# B&R Automation Studio project VInRoS_BaR_AS_Program (part 2)

#### Main.c
```c
#include <bur/plctypes.h>
#include <standard.h>

#ifdef _DEFAULT_INCLUDES
#include <AsDefault.h>
#endif

#include "Main.h"

_LOCAL struct MpAxisBasic MpAxisBasic_0;
_LOCAL struct MpAxisBasicParType AxisParameters;
_LOCAL enum Mechanism_State_ID_enum state_id;

void _INIT ProgramInit(void)
{
	memset(&Global_VInRoS_Str.Mech_Id_3, 0, sizeof(Global_VInRoS_Str.Mech_Id_3));

	MpAxisBasic_0.Enable     = 1;
	MpAxisBasic_0.MpLink     = &gAxis_Mech_03;
	MpAxisBasic_0.Parameters = &AxisParameters;

	Trajectory_Str.Targets.Position[0] = 700.0;
	Trajectory_Str.Targets.Position[1] = 100.0;
	Trajectory_Str.Targets.Position[2] = 400.0;
	Trajectory_Str.Targets.Position[3] = 600.0;
	Trajectory_Str.Targets.Position[4] = 300.0;

	Trajectory_Str.Targets.Velocity[0] = 400.0;
	Trajectory_Str.Targets.Velocity[1] = 200.0;
	Trajectory_Str.Targets.Velocity[2] = 400.0;
	Trajectory_Str.Targets.Velocity[3] = 100.0;
	Trajectory_Str.Targets.Velocity[4] = 400.0;

	Trajectory_Str.Length = 5;

	state_id = MECH_STATE_ACTIVE;
}

void _CYCLIC ProgramCyclic(void)
{
	switch(state_id){
		case MECH_STATE_ACTIVE:
			{
				if(Global_VInRoS_Str.Mech_Id_3.Info.Active == 1){
					state_id = MECH_STATE_POWER;
				}
			}
			break;

		case MECH_STATE_POWER:
			{
				if(Global_VInRoS_Str.Mech_Id_3.Info.Power == 1){
					state_id = MECH_STATE_HOME;
				}
			}
			break;

		case MECH_STATE_HOME:
			{
				if(Global_VInRoS_Str.Mech_Id_3.Info.Home == 1){
					MpAxisBasic_0.Home = 0;
					Global_VInRoS_Str.Mech_Id_3.Command.Home = 0;
					state_id = MECH_STATE_WAIT;
				}
			}
			break;

		case MECH_STATE_WAIT:
			{
				if(Global_VInRoS_Str.Mech_Id_3.Command.Home == 1){
					state_id = MECH_STATE_HOME_UPD_PARAMETERS;
				}

				if(Global_VInRoS_Str.Mech_Id_3.Command.Start == 1){
					Trajectory_Str.Iteration = 0;
					state_id = MECH_STATE_UPD_PARAMETERS;
				}
			}
			break;

		case MECH_STATE_UPD_PARAMETERS:
			{
				Global_VInRoS_Str.Mech_Id_3.Parameters.Position = Trajectory_Str.Targets.Position[Trajectory_Str.Iteration];
				Global_VInRoS_Str.Mech_Id_3.Parameters.Velocity = Trajectory_Str.Targets.Velocity[Trajectory_Str.Iteration];
				Global_VInRoS_Str.Mech_Id_3.Parameters.Acc_Dec  = Trajectory_Str.Targets.Velocity[Trajectory_Str.Iteration]*10;

				Global_VInRoS_Str.Mech_Id_3.Command.Update = 1;
				if(Global_VInRoS_Str.Mech_Id_3.Info.Update_Done == 1){
					state_id = MECH_STATE_MOTION_1;
				}
			}
			break;

		case MECH_STATE_MOTION_1:
			{
				Global_VInRoS_Str.Mech_Id_3.Command.Move = 1;
				if(Global_VInRoS_Str.Mech_Id_3.Info.Move_Active == 1){
					state_id = MECH_STATE_MOTION_2;
				}
			}
			break;

		case MECH_STATE_MOTION_2:
			{
				if(Global_VInRoS_Str.Mech_Id_3.Command.Stop == 1){
					state_id = MECH_STATE_STOP;
				}else{
					if(Global_VInRoS_Str.Mech_Id_3.Info.In_Position == 1){
						Global_VInRoS_Str.Mech_Id_3.Command.Move = 0;

						if(Trajectory_Str.Iteration == Trajectory_Str.Length - 1){
							state_id = MECH_STATE_WAIT;
						}else{
							Trajectory_Str.Iteration++;
							state_id = MECH_STATE_UPD_PARAMETERS;
						}
					}
				}
			}
			break;

		case MECH_STATE_HOME_UPD_PARAMETERS:
			{
				Global_VInRoS_Str.Mech_Id_3.Parameters.Position = 400.0;
				Global_VInRoS_Str.Mech_Id_3.Parameters.Velocity = 250.0;
				Global_VInRoS_Str.Mech_Id_3.Parameters.Acc_Dec  = 2500.0;

				Global_VInRoS_Str.Mech_Id_3.Command.Update = 1;
				if(Global_VInRoS_Str.Mech_Id_3.Info.Update_Done == 1){
					state_id = MECH_STATE_HOME_MOTION_1;
				}
			}
			break;

		case MECH_STATE_HOME_MOTION_1:
			{
				Global_VInRoS_Str.Mech_Id_3.Command.Move = 1;
				if(Global_VInRoS_Str.Mech_Id_3.Info.Move_Active == 1){
					state_id = MECH_STATE_HOME_MOTION_2;
				}
			}
			break;

		case MECH_STATE_HOME_MOTION_2:
			{
				if(Global_VInRoS_Str.Mech_Id_3.Info.In_Position == 1){
					Global_VInRoS_Str.Mech_Id_3.Command.Move = 0;
					Global_VInRoS_Str.Mech_Id_3.Command.Home = 0;
					state_id = MECH_STATE_WAIT;
				}
			}
			break;

		case MECH_STATE_STOP:
			{
				Global_VInRoS_Str.Mech_Id_3.Command.Stop  = 0;
				Global_VInRoS_Str.Mech_Id_3.Command.Start = 0;

				Global_VInRoS_Str.Mech_Id_3.Command.Move = 0;
				if(Global_VInRoS_Str.Mech_Id_3.Info.Move_Active == 0){
					state_id = MECH_STATE_WAIT;
				}
			}
			break;

		case MECH_STATE_SAFETY:
			{
			}
			break;

		case MECH_STATE_ERROR:
			{
				Global_VInRoS_Str.Mech_Id_3.Command.Home   = 0;
				Global_VInRoS_Str.Mech_Id_3.Command.Update = 0;
				Global_VInRoS_Str.Mech_Id_3.Command.Stop   = 0;
				Global_VInRoS_Str.Mech_Id_3.Command.Start  = 0;
				Global_VInRoS_Str.Mech_Id_3.Command.Move   = 0;

				Global_VInRoS_Str.Mech_Id_3.Command.Move = 0;
				if(Global_VInRoS_Str.Mech_Id_3.Info.Error == 0){
					state_id = MECH_STATE_WAIT;
				}
			}
			break;

	}

	AxisParameters.Position     = Global_VInRoS_Str.Mech_Id_3.Parameters.Position;
	AxisParameters.Velocity     = Global_VInRoS_Str.Mech_Id_3.Parameters.Velocity;
	AxisParameters.Acceleration = Global_VInRoS_Str.Mech_Id_3.Parameters.Acc_Dec;
	AxisParameters.Deceleration = Global_VInRoS_Str.Mech_Id_3.Parameters.Acc_Dec;

	MpAxisBasic_0.Power = Global_VInRoS_Str.Mech_Id_3.Command.Power;
	if(Global_VInRoS_Str.Mech_Id_3.Command.Home == 1 && Global_VInRoS_Str.Mech_Id_3.Info.Home == 0){
		MpAxisBasic_0.Home = 1;
	}
	MpAxisBasic_0.ErrorReset = Global_VInRoS_Str.Mech_Id_3.Command.Reset_Error;
	MpAxisBasic_0.Update     = Global_VInRoS_Str.Mech_Id_3.Command.Update;
	MpAxisBasic_0.MoveAbsolute = Global_VInRoS_Str.Mech_Id_3.Command.Move;

	MpAxisBasic(&MpAxisBasic_0);

	Global_VInRoS_Str.Mech_Id_3.Info.Active = MpAxisBasic_0.Active;
	Global_VInRoS_Str.Mech_Id_3.Info.Power  = MpAxisBasic_0.PowerOn;
	Global_VInRoS_Str.Mech_Id_3.Info.Home   = MpAxisBasic_0.IsHomed;
	Global_VInRoS_Str.Mech_Id_3.Info.Error  = MpAxisBasic_0.Error;
	Global_VInRoS_Str.Mech_Id_3.Info.Update_Done = MpAxisBasic_0.UpdateDone;
	Global_VInRoS_Str.Mech_Id_3.Info.Move_Active = MpAxisBasic_0.MoveActive;
	if(MpAxisBasic_0.InPosition == 1 && MpAxisBasic_0.MoveDone == 1){
		Global_VInRoS_Str.Mech_Id_3.Info.In_Position = 1;
	}else{
		Global_VInRoS_Str.Mech_Id_3.Info.In_Position = 0;
	}
	Global_VInRoS_Str.Mech_Id_3.Position = MpAxisBasic_0.Position;

	if(Global_VInRoS_Str.Mech_Id_3.Info.Error == 1){
		state_id = MECH_STATE_ERROR;
	}

	if(SAFETY_ACTIVE == 0 || SAFETY_STATUS == 0){
		Global_VInRoS_Str.Mech_Id_3.Info.Safety = 1;
	}else{
		Global_VInRoS_Str.Mech_Id_3.Info.Safety = 0;
	}
	if(SAFETY_ACTIVE == 1 || SAFETY_STATUS == 0){
		RESET_SAFETY = Global_VInRoS_Str.Mech_Id_3.Command.Reset_Safety;
	}
}
```

### Program Logical/T_EX600 (ANSIC)

#### Main.h
```c
#include <bur/plctypes.h>

#ifdef _DEFAULT_INCLUDES
	#include <AsDefault.h>
#endif

typedef enum EX600_State_ID_enum{
	EX600_STATE_ACTIVE,
	EX600_STATE_HOME,
	EX600_STATE_WAIT,
	EX600_STATE_ERROR
}EX600_State_ID_enum;
```

#### Main.c
```c
// Include B&R Automation libraries (declarations for B&R ANSI C extensions).
#include <bur/plctypes.h>

#ifdef _DEFAULT_INCLUDES
	#include <AsDefault.h>
#endif

#include <Main.h>

// Custom Lib.: Base conversion between data.
#include <Converter.h>

/*  Local Variables.  */
_LOCAL enum EX600_State_ID_enum state_id;

_LOCAL struct Convert_BOOL_Array_To_USINT C_BOOL_Arr_To_USINT_1;
_LOCAL struct Convert_USINT_To_BOOL_Array C_USINT_To_BOOL_Arr_1;
_LOCAL struct Convert_USINT_To_BOOL_Array C_USINT_To_BOOL_Arr_2;

/**
 * Program Intitialization
 */
void _INIT ProgramInit(void)
{
	memset(&Global_VInRoS_Str.EX_600, 0, sizeof(Global_VInRoS_Str.EX_600));

	state_id = EX600_STATE_ACTIVE;
}

/**
 * Program Cyclic
 *
 * Duration (Cycle Time): 10000 [ms]
 * Tolerance            : 10000 [ms]
 */
void _CYCLIC ProgramCyclic(void)
{
	switch(state_id){
		case EX600_STATE_ACTIVE:
			{
				if(Global_VInRoS_Str.EX_600.Slave.Info.Active == 1){
					state_id = EX600_STATE_HOME;
				}
			}
			break;

		case EX600_STATE_HOME:
			{
				if(Global_VInRoS_Str.EX_600.Slave.Command.Home == 1){
					memset(C_BOOL_Arr_To_USINT_1.INPUT, 0, sizeof(C_BOOL_Arr_To_USINT_1.INPUT));
					C_USINT_To_BOOL_Arr_1.INPUT = 0;
					C_USINT_To_BOOL_Arr_2.INPUT = 0;

					Global_VInRoS_Str.EX_600.Slave.Info.Home = 1;
					Global_VInRoS_Str.EX_600.Slave.Command.Home = 0;
					state_id = EX600_STATE_WAIT;
				}
			}
			break;

		case EX600_STATE_WAIT:
			{
				int i;
				for(i = 0; i < (int)(sizeof(C_BOOL_Arr_To_USINT_1.INPUT)/sizeof(C_BOOL_Arr_To_USINT_1.INPUT[0])); i++){
					C_BOOL_Arr_To_USINT_1.INPUT[i] = Global_VInRoS_Str.EX_600.Slave.Output[i];
				}
				Convert_BOOL_Array_To_USINT(&C_BOOL_Arr_To_USINT_1);

				Convert_USINT_To_BOOL_Array(&C_USINT_To_BOOL_Arr_1);
				int j;
				for(j = 0; j < (int)(sizeof(C_USINT_To_BOOL_Arr_1.OUTPUT)/sizeof(C_USINT_To_BOOL_Arr_1.OUTPUT[0])); j++){
					Global_VInRoS_Str.EX_600.Slave.Input[j] = C_USINT_To_BOOL_Arr_1.OUTPUT[j];
				}
				Convert_USINT_To_BOOL_Array(&C_USINT_To_BOOL_Arr_2);
				int k;
				for(k = 0; k < (int)(sizeof(C_USINT_To_BOOL_Arr_2.OUTPUT)/sizeof(C_USINT_To_BOOL_Arr_2.OUTPUT[0])); k++){
					Global_VInRoS_Str.EX_600.Slave.Input[k + 8] = C_USINT_To_BOOL_Arr_2.OUTPUT[k];
				}

			}
			break;

		case EX600_STATE_ERROR:
			{
				if(Global_VInRoS_Str.EX_600.Slave.Info.Error == 0){
					state_id = EX600_STATE_WAIT;
				}
			}
			break;
	}

	if(Global_VInRoS_Str.EX_600.Slave.Info.Error == 1){
		state_id = EX600_STATE_ERROR;
	}
}
```

### Program Logical/T_ROB_1 (ANSIC)

#### Main.c - Init, cyclic, exit code
```c
#include <bur/plctypes.h>

#ifdef _DEFAULT_INCLUDES
#include <AsDefault.h>
#endif

#include <Main.h>

_LOCAL enum Robot_State_ID_enum state_id;

/*
if(Global_VInRoS_Str.Rob_Id_1.Command.Start == TRUE){
	ABB_Library_Rob_1.Command.ID.Motion = MAIN_ID_JOINT_ABSOLUTE;
	ABB_Library_Rob_1.Command.START = TRUE;
	Global_VInRoS_Str.Rob_Id_1.Command.Start = FALSE;
}
   */

/*
if(Global_VInRoS_Str.Rob_Id_1.Command.STOP == TRUE){
	ABB_Library_Rob_1.Command.STOP = TRUE;
	Global_VInRoS_Str.Rob_Id_1.Command.STOP = FALSE;
}
*/

void _INIT ProgramInit(void)
{
	memset(&Global_VInRoS_Str.Rob_Id_1, 0, sizeof(Global_VInRoS_Str.Rob_Id_1));

	ABB_Library_Rob_1.Enable = TRUE;

	//
	ABB_Library_Rob_1.Rob_Tool.robHold = FALSE;
	ABB_Library_Rob_1.Rob_Tool.tFrame.Position[0] = 0.0; ABB_Library_Rob_1.Rob_Tool.tFrame.Position[1] = 0.0;
	ABB_Library_Rob_1.Rob_Tool.tFrame.Position[2] = 0.0;
	ABB_Library_Rob_1.Rob_Tool.tFrame.Rotation[0] = 1.0; ABB_Library_Rob_1.Rob_Tool.tFrame.Rotation[1] = 0.0;
	ABB_Library_Rob_1.Rob_Tool.tFrame.Rotation[2] = 0.0; ABB_Library_Rob_1.Rob_Tool.tFrame.Rotation[3] = 0.0;
	ABB_Library_Rob_1.Rob_Tool.tLoad.mass = 0.0;
	ABB_Library_Rob_1.Rob_Tool.tLoad.center_of_gravity[0] = 0.0; ABB_Library_Rob_1.Rob_Tool.tLoad.center_of_gravity[1] = 0.0;
	ABB_Library_Rob_1.Rob_Tool.tLoad.center_of_gravity[2] = 0.0;
	ABB_Library_Rob_1.Rob_Tool.tLoad.intertial_axes[0] = 1.0; ABB_Library_Rob_1.Rob_Tool.tLoad.intertial_axes[1] = 0.0;
	ABB_Library_Rob_1.Rob_Tool.tLoad.intertial_axes[2] = 0.0; ABB_Library_Rob_1.Rob_Tool.tLoad.intertial_axes[3] = 0.0;
	ABB_Library_Rob_1.Rob_Tool.tLoad.moment_of_inertia[0] = 0.0; ABB_Library_Rob_1.Rob_Tool.tLoad.moment_of_inertia[1] = 0.0;
	ABB_Library_Rob_1.Rob_Tool.tLoad.moment_of_inertia[2] = 0.0;

	ABB_Library_Rob_1.Parameter.Joint[0].Q[0] = 130.0; ABB_Library_Rob_1.Parameter.Joint[0].Q[1] = -10.0;
	ABB_Library_Rob_1.Parameter.Joint[0].Q[2] = 15.0; ABB_Library_Rob_1.Parameter.Joint[0].Q[3] = -50.0;
	ABB_Library_Rob_1.Parameter.Joint[0].Q[4] = 60.0; ABB_Library_Rob_1.Parameter.Joint[0].Q[5] = 60.0;
	ABB_Library_Rob_1.Parameter.Speed[0] = vSPEED_100;
	ABB_Library_Rob_1.Parameter.Zone[0]  = zZone_fine;

	ABB_Library_Rob_1.Parameter.Joint[1].Q[0] = 110.0; ABB_Library_Rob_1.Parameter.Joint[1].Q[1] = 60.0;
	ABB_Library_Rob_1.Parameter.Joint[1].Q[2] = -20.0; ABB_Library_Rob_1.Parameter.Joint[1].Q[3] = 0.0;
	ABB_Library_Rob_1.Parameter.Joint[1].Q[4] = -60.0; ABB_Library_Rob_1.Parameter.Joint[1].Q[5] = -40.0;
	ABB_Library_Rob_1.Parameter.Speed[1] = vSPEED_100;
	ABB_Library_Rob_1.Parameter.Zone[1]  = zZone_fine;

	ABB_Library_Rob_1.Parameter.Joint[2].Q[0] = -30.0; ABB_Library_Rob_1.Parameter.Joint[2].Q[1] = 20.0;
	ABB_Library_Rob_1.Parameter.Joint[2].Q[2] = 10.0; ABB_Library_Rob_1.Parameter.Joint[2].Q[3] = 40.0;
	ABB_Library_Rob_1.Parameter.Joint[2].Q[4] = 90.0; ABB_Library_Rob_1.Parameter.Joint[2].Q[5] = 0.0;
	ABB_Library_Rob_1.Parameter.Speed[2] = vSPEED_100;
	ABB_Library_Rob_1.Parameter.Zone[2]  = zZone_fine;

	ABB_Library_Rob_1.Parameter.Joint[3].Q[0] = 0.0; ABB_Library_Rob_1.Parameter.Joint[3].Q[1] = -50.0;
	ABB_Library_Rob_1.Parameter.Joint[3].Q[2] = -20.0; ABB_Library_Rob_1.Parameter.Joint[3].Q[3] = 90.0;
	ABB_Library_Rob_1.Parameter.Joint[3].Q[4] = -40.0; ABB_Library_Rob_1.Parameter.Joint[3].Q[5] = 100.0;
	ABB_Library_Rob_1.Parameter.Speed[3] = vSPEED_100;
	ABB_Library_Rob_1.Parameter.Zone[3]  = zZone_fine;

	ABB_Library_Rob_1.Parameter.Joint[4].Q[0] = 65.0; ABB_Library_Rob_1.Parameter.Joint[4].Q[1] = 10.0;
	ABB_Library_Rob_1.Parameter.Joint[4].Q[2] = 20.0; ABB_Library_Rob_1.Parameter.Joint[4].Q[3] = 50.0;
	ABB_Library_Rob_1.Parameter.Joint[4].Q[4] = 55.0; ABB_Library_Rob_1.Parameter.Joint[4].Q[5] = -20.0;
	ABB_Library_Rob_1.Parameter.Speed[4] = vSPEED_100;
	ABB_Library_Rob_1.Parameter.Zone[4]  = zZone_fine;

	ABB_Library_Rob_1.Parameter.Trajectory_Size = 5;

	/*
	ABB_Library_Rob_1.Parameter.TCP[0].Position[0] = 0.0; ABB_Library_Rob_1.Parameter.TCP[0].Position[1] = 0.0;
	ABB_Library_Rob_1.Parameter.TCP[0].Position[2] = 0.0;
	ABB_Library_Rob_1.Parameter.TCP[0].Rotation[0] = 0.0; ABB_Library_Rob_1.Parameter.TCP[0].Rotation[1] = 0.0;
	ABB_Library_Rob_1.Parameter.TCP[0].Rotation[2] = 0.0;
	ABB_Library_Rob_1.Parameter.TCP[0].Configuration[0] = 0.0; ABB_Library_Rob_1.Parameter.TCP[0].Configuration[1] = 0.0;
	ABB_Library_Rob_1.Parameter.TCP[0].Configuration[2] = 0.0; ABB_Library_Rob_1.Parameter.TCP[0].Configuration[3] = 0.0;
	ABB_Library_Rob_1.Parameter.Speed[0] = 8;
	ABB_Library_Rob_1.Parameter.Zone[0]  = 0;

	ABB_Library_Rob_1.Parameter.Trajectory_Size = 2;
	*/

	/*
	//
	Trajectory_Str.Targets.Position[0].Q[0] = 0.0; Trajectory_Str.Targets.Position[0].Q[1] = 0.0;
	Trajectory_Str.Targets.Position[0].Q[2] = 0.0; Trajectory_Str.Targets.Position[0].Q[3] = 0.0;
	Trajectory_Str.Targets.Position[0].Q[4] = 0.0; Trajectory_Str.Targets.Position[0].Q[5] = 0.0;
	Trajectory_Str.Targets.Speed[0] = 8;
	Trajectory_Str.Targets.Zone[0]  = 0;
	//
	Trajectory_Str.Targets.Position[1].Q[0] = 0.0; Trajectory_Str.Targets.Position[1].Q[1] = 0.0;
	Trajectory_Str.Targets.Position[1].Q[2] = 0.0; Trajectory_Str.Targets.Position[1].Q[3] = 0.0;
	Trajectory_Str.Targets.Position[1].Q[4] = 90.0; Trajectory_Str.Targets.Position[1].Q[5] = 0.0;
	Trajectory_Str.Targets.Speed[1] = 8;
	Trajectory_Str.Targets.Zone[1]  = 0;
	//
	Trajectory_Str.Targets.Position[2].Q[0] = 90.0; Trajectory_Str.Targets.Position[2].Q[1] = 0.0;
	Trajectory_Str.Targets.Position[2].Q[2] = 0.0; Trajectory_Str.Targets.Position[2].Q[3] = 0.0;
	Trajectory_Str.Targets.Position[2].Q[4] = 90.0; Trajectory_Str.Targets.Position[2].Q[5] = 0.0;
	Trajectory_Str.Targets.Speed[2] = 8;
	Trajectory_Str.Targets.Zone[2]  = 0;
	//
	Trajectory_Str.Targets.Position[3].Q[0] = 90.0; Trajectory_Str.Targets.Position[3].Q[1] = 0.0;
	Trajectory_Str.Targets.Position[3].Q[2] = 0.0; Trajectory_Str.Targets.Position[3].Q[3] = 45.0;
	Trajectory_Str.Targets.Position[3].Q[4] = 90.0; Trajectory_Str.Targets.Position[3].Q[5] = 0.0;
	Trajectory_Str.Targets.Speed[3] = 8;
	Trajectory_Str.Targets.Zone[3]  = 0;
	//
	Trajectory_Str.Targets.Position[4].Q[0] = 0.0; Trajectory_Str.Targets.Position[4].Q[1] = 0.0;
	Trajectory_Str.Targets.Position[4].Q[2] = 0.0; Trajectory_Str.Targets.Position[4].Q[3] = 45.0;
	Trajectory_Str.Targets.Position[4].Q[4] = 90.0; Trajectory_Str.Targets.Position[4].Q[5] = 0.0;
	Trajectory_Str.Targets.Speed[4] = 8;
	Trajectory_Str.Targets.Zone[4]  = 0;

	//
	Trajectory_Str.Length = 5;
	*/
}

void _CYCLIC ProgramCyclic(void)
{
	/*
	switch(state_id){
		case ROB_STATE_ACTIVE:
			{
				if(Global_VInRoS_Str.Rob_Id_1.Info.Active == TRUE){
					state_id = ROB_STATE_POWER;
				}
			}
			break;

		case ROB_STATE_POWER:
			{
				if(Global_VInRoS_Str.Rob_Id_1.Info.Power == TRUE){
					state_id = ROB_STATE_WAIT;
				}
			}
			break;

		case ROB_STATE_WAIT:
			{
				Global_VInRoS_Str.Rob_Id_1.Info.Move_Active = FALSE;

				if(Global_VInRoS_Str.Rob_Id_1.Command.Home == TRUE){
					state_id = ROB_STATE_UPD_PARAMETERS;
				}

				if(Global_VInRoS_Str.Rob_Id_1.Command.Start == TRUE){
					Trajectory_Str.Iteration = FALSE;
					state_id = ROB_STATE_HOME_UPD_PARAMETERS;
				}
			}
			break;

		case ROB_STATE_UPD_PARAMETERS:
			{
				memcpy(ABB_Library_Rob_1.Parameter.Position, Trajectory_Str.Targets.Position,
					  (sizeof(Trajectory_Str.Targets.Position) / sizeof(Trajectory_Str.Targets.Position[0])) * sizeof(REAL));
				memcpy(ABB_Library_Rob_1.Parameter.Speed, Trajectory_Str.Targets.Speed,
					   (sizeof(Trajectory_Str.Targets.Speed) / sizeof(Trajectory_Str.Targets.Speed[0])) * sizeof(REAL));
				memcpy(ABB_Library_Rob_1.Parameter.Zone, Trajectory_Str.Targets.Zone,
					   (sizeof(Trajectory_Str.Targets.Zone) / sizeof(Trajectory_Str.Targets.Zone[0])) * sizeof(REAL));

				ABB_Library_Rob_1.Parameter.Trajectory_Size = Trajectory_Str.Length;

				Global_VInRoS_Str.Rob_Id_1.Command.Update = TRUE;

				if(Global_VInRoS_Str.Rob_Id_1.Info.Update_Done == TRUE){
					state_id = ROB_STATE_MOTION_1;
				}
			}
			break;

		case ROB_STATE_MOTION_1:
			{
				Global_VInRoS_Str.Rob_Id_1.Info.Move_Active = TRUE;
			}
			break;

		case ROB_STATE_MOTION_2:
			{

			}
			break;

		case ROB_STATE_HOME_UPD_PARAMETERS:
			{
				Global_VInRoS_Str.Rob_Id_1.Info.Home = FALSE;

				ABB_Library_Rob_1.Parameter.Position[0].Q[0] = 0.0; ABB_Library_Rob_1.Parameter.Position[0].Q[1] = 0.0;
				ABB_Library_Rob_1.Parameter.Position[0].Q[2] = 0.0; ABB_Library_Rob_1.Parameter.Position[0].Q[3] = 0.0;
				ABB_Library_Rob_1.Parameter.Position[0].Q[4] = 0.0; ABB_Library_Rob_1.Parameter.Position[0].Q[5] = 0.0;
				ABB_Library_Rob_1.Parameter.Speed[0] = 5;
				ABB_Library_Rob_1.Parameter.Zone[0]  = 0;

				ABB_Library_Rob_1.Parameter.Trajectory_Size = 1;

				Global_VInRoS_Str.Rob_Id_1.Command.Update = TRUE;

				if(Global_VInRoS_Str.Rob_Id_1.Info.Update_Done == TRUE){
					state_id = ROB_STATE_HOME_MOTION_1;
				}
			}
			break;

		case ROB_STATE_HOME_MOTION_1:
			{

			}
			break;

		case ROB_STATE_HOME_MOTION_2:
			{
				Global_VInRoS_Str.Rob_Id_1.Info.Home = TRUE;
			}
			break;

		case ROB_STATE_STOP:
			{
				Global_VInRoS_Str.Rob_Id_1.Info.Move_Active = FALSE;
			}
			break;

		case ROB_STATE_SAFETY:
			{

			}
			break;

		case ROB_STATE_ERROR:
			{

			}
			break;
	}

	if(Global_VInRoS_Str.Rob_Id_1.Command.Update == TRUE){
		ABB_Library_Rob_1.Command.ID.Update = UPT_ID_TRAJECTORY_JOINT;
		ABB_Library_Rob_1.Command.UPDATE = TRUE;
		Global_VInRoS_Str.Rob_Id_1.Command.Update = FALSE;
	}

	ABB_Library(&ABB_Library_Rob_1);

	Global_VInRoS_Str.Rob_Id_1.Info.Active = ABB_Library_Rob_1.Status.Robot.Active;
	Global_VInRoS_Str.Rob_Id_1.Info.Power = ABB_Library_Rob_1.Status.Robot.System.MOTOR_ON;
	Global_VInRoS_Str.Rob_Id_1.Info.Update_Done = ABB_Library_Rob_1.Status.Robot.Update_Done;
	Global_VInRoS_Str.Rob_Id_1.Info.In_Position = ABB_Library_Rob_1.Status.Robot.In_Position;
	Global_VInRoS_Str.Rob_Id_1.Info.Error  = FALSE;
	Global_VInRoS_Str.Rob_Id_1.Info.Safety = FALSE;

	memcpy(Global_VInRoS_Str.Rob_Id_1.Position.Q, ABB_Library_Rob_1.RT_Data.Q,
		(sizeof(ABB_Library_Rob_1.RT_Data.Q) / sizeof(ABB_Library_Rob_1.RT_Data.Q[0])) * sizeof(REAL));

	if(Global_VInRoS_Str.Rob_Id_1.Info.Error == TRUE){
		state_id = ROB_STATE_ERROR;
	}

	if(SAFETY_ACTIVE == FALSE || SAFETY_STATUS == FALSE){
		Global_VInRoS_Str.Rob_Id_1.Info.Safety = TRUE;
	}else{
		Global_VInRoS_Str.Rob_Id_1.Info.Safety = FALSE;
	}
	if(SAFETY_ACTIVE == TRUE || SAFETY_STATUS == FALSE){
		RESET_SAFETY = Global_VInRoS_Str.Rob_Id_1.Command.Reset_Safety;
	}
*/

	ABB_Library(&ABB_Library_Rob_1);
}
```

#### Main.h - Init, cyclic, exit code
```c
#include <bur/plctypes.h>

#ifdef _DEFAULT_INCLUDES
#include <AsDefault.h>
#endif

#include "ABB_Library.h"

// Custom Lib.: Base conversion between data.
#include "Converter.h"

_LOCAL struct ABB_Library ABB_Library_Rob_1;

_LOCAL USINT PROFINET_Mapping_IN[256];
_LOCAL USINT PROFINET_Mapping_OUT[256];
```

#### ABB_Library.h - Init, cyclic, exit code
```c
#ifndef HEADER_FILE_ABB_LIBRARY
#define HEADER_FILE_ABB_LIBRARY

// Include B&R Automation libraries (declarations for B&R ANSI C extensions).
#include <bur/plctypes.h>

// Custom Lib.: Base conversion between data.
#include "Converter.h"

// Include other libraries.
#include <math.h>

// Directive (macro definition).
#ifndef M_PI
#define M_PI 3.14159265358979323846264338327950288
#endif

#define DegToRad(value) ((value) * M_PI / 180.0)
#define RadToDeg(value) ((value) * 180.0 / M_PI)

#define TRUE 1
#define FALSE (!TRUE)
#define NULL 0
#define CEIL_DEFUALT_FACTOR 10

_LOCAL UINT aux_trajectory_ID;

typedef enum ABB_Library_statesPLC_enum{
	ABBt_STATE_INITIALIZATION     = 0,
	ABBt_STATE_START_INIT         = 5,
	ABBt_STATE_START_MOTOR_ON     = 6,
	ABBt_STATE_START_PP_TO_M      = 7,
	ABBt_STATE_START_EXECUTE      = 8,
	ABBt_STATE_STOP_INIT          = 10,
	ABBt_STATE_STOP_EXECUTE       = 11,
	ABBt_STATE_STOP_MOTOR_OFF     = 12,
	ABBt_STATE_STOPPED_PP_TO_MAIN = 13,
	ABBt_STATE_STOPPED_TO_START   = 14,
	ABBt_STATE_WAIT               = 20,
	ABBt_STATE_MOVE_JOINT_CHECK   = 30,
	ABBt_STATE_MOVE_JOINT_EXECUTE = 31,
	ABBt_STATE_MOVE_TCP_CHECK     = 40,
	ABBt_STATE_MOVE_TCP_EXECUTE   = 41
}ABB_Library_statesPLC_enum;

typedef enum ABB_Library_statesROB_m_enum{
	ABBr_STATE_INITIALIZATION = 10,
	ABBr_STATE_WAIT           = 20,
	ABBr_STATE_MOVE_JOINT     = 30,
	ABBr_STATE_MOVE_TCP       = 40
}ABB_Library_statesROB_m_enum;

typedef enum ABB_Library_statesROB_u_enum{
	ABBu_STATE_INITIALIZATION      = 10,
	ABBu_STATE_UPDATE_JOINT_TRAJ_1 = 40,
	ABBu_STATE_UPDATE_JOINT_TRAJ_2 = 41,
	ABBu_STATE_UPDATE_JOINT_TRAJ_3 = 42,
	ABBu_STATE_UPDATE_JOINT_TRAJ_4 = 43,
	ABBu_STATE_UPDATE_TCP_TRAJ_1   = 50,
	ABBu_STATE_UPDATE_TCP_TRAJ_2   = 51,
	ABBu_STATE_UPDATE_TCP_TRAJ_3   = 52,
	ABBu_STATE_UPDATE_TCP_TRAJ_4   = 53,
	ABBu_STATE_UPDATE_TOOL_PARAM   = 100
}ABB_Library_statesROB_u_enum;

typedef enum ABB_Library_cmd_m_state_enum{
	MAIN_ID_EMPTY		   = 0,
	MAIN_ID_JOINT_ABSOLUTE = 1,
	MAIN_ID_TCP_LINEAR     = 2,
}ABB_Library_cmd_m_state_enum;

typedef enum ABB_Library_cmd_u_state_enum{
	UPT_ID_EMPTY			= 0,
	UPT_ID_TRAJECTORY_JOINT = 1,
	UPT_ID_TRAJECTORY_TCP   = 2,
	UPT_ID_ROB_TOOL	        = 10
}ABB_Library_cmd_u_state_enum;

typedef enum ABB_Library_update_enum{
	UPT_STATE_INITIALIZATION = 0,
	UPT_STATE_WAIT           = 10,
	UPT_STATE_JOINT_TRAJ_1   = 40,
	UPT_STATE_JOINT_TRAJ_2   = 41,
	UPT_STATE_JOINT_TRAJ_3   = 42,
	UPT_STATE_JOINT_TRAJ_4   = 43,
	UPT_STATE_TCP_TRAJ_1     = 50,
	UPT_STATE_TCP_TRAJ_2     = 51,
	UPT_STATE_TCP_TRAJ_3     = 52,
	UPT_STATE_TCP_TRAJ_4     = 53,
	UPT_STATE_RTOOL          = 100
}ABB_Library_update_enum;

typedef enum ABB_Library_mParam_speed_enum{
	vSPEED_5,
	vSPEED_10,
	vSPEED_20,
	vSPEED_30,
	vSPEED_40,
	vSPEED_50,
	vSPEED_60,
	vSPEED_80,
	vSPEED_100,
	vSPEED_150,
	vSPEED_200,
	vSPEED_300,
	vSPEED_400,
	vSPEED_500,
	vSPEED_600,
	vSPEED_800,
	vSPEED_1000,
	vSPEED_1500,
	vSPEED_2000,
	vSPEED_2500,
	vSPEED_3000,
	vSPEED_4000,
	vSPEED_5000,
	vSPEED_6000
}ABB_Library_mParam_speed_enum;

typedef enum ABB_Library_mParam_zone_enum{
	zZone_fine,
	zZone_0,
	zZone_1,
	zZone_5,
	zZone_10,
	zZone_15,
	zZone_20,
	zZone_30,
	zZone_40,
	zZone_50,
	zZone_60,
	zZone_80,
	zZone_100,
	zZone_150,
	zZone_200
}ABB_Library_mParam_zone_enum;

typedef struct ABB_Library_internal_update_str{
	UINT ID;
	ABB_Library_update_enum actual_state;
}ABB_Library_internal_update_str;

typedef struct ABB_Library_internal_str{
	ABB_Library_statesPLC_enum actual_state;
	ABB_Library_statesPLC_enum before_state;
	ABB_Library_internal_update_str Update;
	REAL ACCURACY_FACTOR;
	REAL ACCURACY_FACTOR_QUATERNION;
}ABB_Library_internal_str;

typedef struct ABB_Library_profinet_in_str{
	struct Convert_USINT_To_BOOL_Array STATUS;
	USINT STATE_mID;
	struct Convert_USINT_To_BOOL_Array SYSTEM;
	USINT STATE_uID;
	struct Convert_USINT_Array_To_UINT MOTION_TRAJECTORY_ID;
	struct Convert_USINT_Array_To_UINT JOINT_POS[7];
	struct Convert_USINT_To_BOOL_Array JOINT_POS_SIGN;
	struct Convert_USINT_Array_To_UDINT TCP_POS[3];
	struct Convert_USINT_Array_To_UINT TCP_ROT[3];
	struct Convert_USINT_Array_To_UINT TCP_EX_POS;
	struct Convert_USINT_To_BOOL_Array TCP_SIGN;
	USINT TCP_CFG[4];
	struct Convert_USINT_To_BOOL_Array TCP_CFG_SIGN;
}ABB_Library_profinet_in_str;

typedef struct ABB_Library_profinet_out_str{
	struct Convert_BOOL_Array_To_USINT STATUS;
	struct Convert_BOOL_Array_To_USINT SYSTEM;
	struct Convert_BOOL_Array_To_USINT COMMAND;
	USINT COMMAND_mID;
	USINT COMMAND_uID;
	struct Convert_UINT_To_USINT_Array TRAJECTORY_SIZE;
	USINT SPEED;
	USINT ZONE;
	struct Convert_UINT_To_USINT_Array JOINT_POS[7];
	struct Convert_BOOL_Array_To_USINT JOINT_POS_SIGN;
	struct Convert_UDINT_To_USINT_Array TCP_POS[3];
	struct Convert_UINT_To_USINT_Array TCP_ROT[3];
	struct Convert_UINT_To_USINT_Array TCP_EX_POS;
	struct Convert_BOOL_Array_To_USINT TCP_SIGN;
	USINT TCP_CFG[4];
	struct Convert_BOOL_Array_To_USINT TCP_CFG_SIGN;
	struct Convert_BOOL_Array_To_USINT RTOOL_RH;
	struct Convert_UINT_To_USINT_Array RTOOL_POS[3];
	struct Convert_BOOL_Array_To_USINT RTOOL_POS_SIGN;
	struct Convert_UDINT_To_USINT_Array RTOOL_ROT_QUAT[4];
	struct Convert_BOOL_Array_To_USINT RTOOL_ROT_QUAT_SIGN;
	struct Convert_UINT_To_USINT_Array RTOOL_MASS;
	struct Convert_UDINT_To_USINT_Array RTOOL_COG[3];
	struct Convert_BOOL_Array_To_USINT RTOOL_COG_SIGN;
	struct Convert_UDINT_To_USINT_Array RTOOL_AOM_QUAT[4];
	struct Convert_BOOL_Array_To_USINT RTOOL_AOM_QUAT_SIGN;
	struct Convert_UDINT_To_USINT_Array RTOOL_MOI[3];
}ABB_Library_profinet_out_str;

typedef struct ABB_Library_sysOUT_str{
	BOOL MOTOR_ON;
	BOOL MOTOR_OFF;
	BOOL PP_TO_MAIN;
	BOOL START;
	BOOL STOP;
}ABB_Library_sysOUT_str;

typedef struct ABB_Library_id_cmd_str{
	ABB_Library_cmd_m_state_enum Motion;
	ABB_Library_cmd_u_state_enum Update;
}ABB_Library_id_cmd_str;

typedef struct ABB_Library_command_str{
	BOOL START;
	BOOL STOP;
	BOOL UPDATE;
	ABB_Library_id_cmd_str ID;
	ABB_Library_sysOUT_str System;
}ABB_Library_command_str;

typedef struct ABB_Library_TCP_str{
	REAL Position[3];
	REAL Rotation[3];
	SINT Configuration[4];
	REAL External_Position;
}ABB_Library_TCP_str;

typedef struct ABB_Library_profinet_rtData_str{
	REAL Q[7];
	ABB_Library_TCP_str TCP;
}ABB_Library_profinet_rtData_str;

typedef struct ABB_Library_profinet_Jw_str{
	REAL Q[7];
}ABB_Library_profinet_Jw_str;

typedef struct ABB_Library_parameter_str{
	ABB_Library_profinet_Jw_str Joint[100];
	ABB_Library_TCP_str TCP[100];
	ABB_Library_mParam_speed_enum Speed[100];
	ABB_Library_mParam_zone_enum Zone[100];
	UINT Trajectory_Size;
}ABB_Library_parameter_str;

typedef struct ABB_Library_rTool_tf_str{
	// Translation part.
	REAL Position[3];
	// Rotation part (Quaternion).
	REAL Rotation[4];
}ABB_Library_rTool_tf_str;

typedef struct ABB_Library_rTool_tl_str{
	// Tool Mass.
	REAL mass;
	// Center of Gravity.
	REAL center_of_gravity[3];
	// Inertial axes of tool load.
	REAL intertial_axes[4];
	// Momets of inertia.
	REAL moment_of_inertia[3];
}ABB_Library_rTool_tl_str;

typedef struct ABB_Library_robTool_str{
	// The robot is holding the tool (TRUE / FALSE).
	BOOL robHold;
	// Tool Frame.
	ABB_Library_rTool_tf_str tFrame;
	// Tool Load.
	ABB_Library_rTool_tl_str tLoad;
}ABB_Library_robTool_str;

typedef struct ABB_Library_statusPLC_str{
	BOOL Active;
	BOOL Module_OK;
	BOOL Update_Done;
}ABB_Library_statusPLC_str;

typedef struct ABB_Library_sysIN_str{
	BOOL MOTOR_ON;
	BOOL MOTOR_OFF;
	BOOL PP_MOVED;
	BOOL CYCLE_ON;
}ABB_Library_sysIN_str;

typedef struct ABB_Library_id_statesROB_str{
	ABB_Library_statesROB_m_enum Motion;
	ABB_Library_statesROB_u_enum Update;
}ABB_Library_id_statesROB_str;

typedef struct ABB_Library_statusROB_str{
	BOOL Active;
	BOOL In_Position;
	ABB_Library_id_statesROB_str ID;
	BOOL Update_Done;
	ABB_Library_sysIN_str System;
	UINT Trajectory_ID;
}ABB_Library_statusROB_str;

typedef struct ABB_Library_status_str{
	ABB_Library_statusPLC_str PLC;
	ABB_Library_statusROB_str Robot;
}ABB_Library_status_str;

typedef struct ABB_Library
{
	/**
	Description:
		Function block ...
	*/

	/**
 	 * FUNCTION BLOCK: ABB_Library
	 * INPUT VARIABLES
 	 */
	BOOL Enable;
	BOOL Power_ON;
	BOOL Power_OFF;
	ABB_Library_command_str Command;
	ABB_Library_parameter_str Parameter;
	ABB_Library_robTool_str Rob_Tool;
	ABB_Library_profinet_in_str PROFINET_Mapping_IN;

	/**
 	 * FUNCTION BLOCK: ABB_Library
	 * OUTPUT VARIABLES
 	 */
	ABB_Library_status_str Status;
	ABB_Library_profinet_out_str PROFINET_Mapping_OUT;
	ABB_Library_profinet_rtData_str RT_Data;

	/**
 	 * FUNCTION BLOCK: ABB_Library
	 * INTERNAL VARIABLES
 	 */
	ABB_Library_internal_str Internal;

} ABB_Library_typ;

/**
 * Declaration of the function block ....
 */
_BUR_PUBLIC void ABB_Library(struct ABB_Library* inst);
void Template_Reset(struct ABB_Library* inst);
void Update_Parameters(struct ABB_Library* inst);
void Read_Data_ROB_to_PLC(struct ABB_Library* inst);
void Write_Data_PLC_to_ROB(struct ABB_Library* inst);

void ABB_Library(struct ABB_Library* inst){
	/**
	Description:
		Function block ...

	Args:
		(1) inst [struct ABB_Library*]: Function block instance.
	*/

	if(inst->Enable != TRUE){
		Template_Reset(inst);
	}else{
		Read_Data_ROB_to_PLC(inst);
	}

	switch(inst->Internal.actual_state){
		case ABBt_STATE_INITIALIZATION:
			{
				inst->Internal.ACCURACY_FACTOR 			    = 100;
				inst->Internal.ACCURACY_FACTOR_QUATERNION   = 100000000;

				if(inst->Status.PLC.Active == TRUE){
					inst->Internal.actual_state = ABBt_STATE_START_INIT;
				}
			}
			break;

		case ABBt_STATE_START_INIT:
			{
				inst->Power_OFF = FALSE;

				memset(&inst->Command.System, NULL, sizeof(inst->Command.System));

				if(inst->Power_ON == TRUE && inst->Status.Robot.System.MOTOR_ON == FALSE){
					inst->Internal.actual_state = ABBt_STATE_START_MOTOR_ON;
				}else if(inst->Power_ON == TRUE && inst->Status.Robot.System.MOTOR_ON == TRUE){
					inst->Internal.actual_state = ABBt_STATE_START_PP_TO_M;
				}
			}
			break;

		case ABBt_STATE_START_MOTOR_ON:
			{
				inst->Command.System.MOTOR_ON = TRUE;

				if(inst->Status.Robot.System.MOTOR_ON == TRUE){
					inst->Command.System.MOTOR_ON = FALSE;
					inst->Internal.actual_state   = ABBt_STATE_START_PP_TO_M;
				}
			}
			break;

		case ABBt_STATE_START_PP_TO_M:
			{
				inst->Command.System.PP_TO_MAIN = TRUE;

				if(inst->Status.Robot.System.PP_MOVED == TRUE){
					inst->Command.System.PP_TO_MAIN = FALSE;
					inst->Internal.actual_state     = ABBt_STATE_START_EXECUTE;
				}
			}
			break;

		case ABBt_STATE_START_EXECUTE:
			{
				inst->Command.System.START = TRUE;

				if(inst->Status.Robot.System.CYCLE_ON == TRUE && inst->Status.Robot.Active == TRUE){
					inst->Command.System.START  = FALSE;
					inst->Internal.actual_state = ABBt_STATE_WAIT;
				}
			}
			break;

		case ABBt_STATE_STOP_EXECUTE:
			{
				inst->Command.System.STOP = TRUE;

				if(inst->Status.Robot.System.CYCLE_ON == FALSE){
					inst->Command.System.STOP   = FALSE;
					if(inst->Power_OFF == TRUE){
						inst->Power_OFF             = FALSE;
						inst->Internal.actual_state = ABBt_STATE_STOP_MOTOR_OFF;
					}else if(inst->Command.STOP == TRUE){
						inst->Command.STOP = FALSE;
						inst->Internal.actual_state = ABBt_STATE_STOPPED_PP_TO_MAIN;
					}
				}
			}
			break;

		case ABBt_STATE_STOP_MOTOR_OFF:
			{
				inst->Command.System.MOTOR_OFF = TRUE;

				if(inst->Status.Robot.System.MOTOR_OFF == TRUE){
					inst->Command.System.MOTOR_OFF = FALSE;
					inst->Internal.actual_state    = ABBt_STATE_START_INIT;
				}
			}
			break;

		case ABBt_STATE_STOPPED_PP_TO_MAIN:
			{
				inst->Command.System.PP_TO_MAIN = TRUE;

				if(inst->Status.Robot.System.PP_MOVED == TRUE){
					inst->Command.System.PP_TO_MAIN = FALSE;
					inst->Internal.actual_state     = ABBt_STATE_STOPPED_TO_START;
				}
			}
			break;

		case ABBt_STATE_STOPPED_TO_START:
			{
				inst->Command.System.START = TRUE;

				if(inst->Status.Robot.System.CYCLE_ON == TRUE && inst->Status.Robot.Active == TRUE){
					inst->Command.System.START  = FALSE;
					inst->Internal.actual_state = ABBt_STATE_WAIT;
				}
			}
			break;

		case ABBt_STATE_WAIT:
			{
				inst->Power_ON = FALSE;

				if(inst->Command.START == TRUE && inst->Command.ID.Motion == MAIN_ID_JOINT_ABSOLUTE){
					inst->Command.STOP          = FALSE;
					inst->Internal.actual_state = ABBt_STATE_MOVE_JOINT_CHECK;
				}else if(inst->Command.START == TRUE && inst->Command.ID.Motion == MAIN_ID_TCP_LINEAR){
					inst->Command.STOP          = FALSE;
					inst->Internal.actual_state = ABBt_STATE_MOVE_TCP_CHECK;
				}

				if(inst->Power_OFF == TRUE){
					inst->Internal.actual_state = ABBt_STATE_STOP_EXECUTE;
				}
			}
			break;

		case ABBt_STATE_MOVE_JOINT_CHECK:
			{
				inst->Internal.before_state = ABBt_STATE_MOVE_JOINT_CHECK;

				if(inst->Status.Robot.ID.Motion == ABBr_STATE_MOVE_JOINT && inst->Status.Robot.In_Position == FALSE){
					inst->Command.START     = FALSE;
					inst->Command.ID.Motion = MAIN_ID_EMPTY;

					inst->Internal.actual_state = ABBt_STATE_MOVE_JOINT_EXECUTE;
				}
			}
			break;

		case ABBt_STATE_MOVE_JOINT_EXECUTE:
			{
				inst->Internal.before_state = ABBt_STATE_MOVE_JOINT_EXECUTE;

				if(inst->Status.Robot.In_Position == TRUE){
					inst->Command.START     = FALSE;
					inst->Command.ID.Motion = MAIN_ID_EMPTY;

					inst->Internal.actual_state = ABBt_STATE_WAIT;
				}
			}
			break;

		case ABBt_STATE_MOVE_TCP_CHECK:
			{
				inst->Internal.before_state = ABBt_STATE_MOVE_TCP_CHECK;

				if(inst->Status.Robot.ID.Motion == ABBr_STATE_MOVE_TCP && inst->Status.Robot.In_Position == FALSE){
					inst->Command.START     = FALSE;
					inst->Command.ID.Motion = MAIN_ID_EMPTY;

					inst->Internal.actual_state = ABBt_STATE_MOVE_TCP_EXECUTE;
				}
			}
			break;

		case ABBt_STATE_MOVE_TCP_EXECUTE:
			{
				inst->Internal.before_state = ABBt_STATE_MOVE_TCP_EXECUTE;

				if(inst->Status.Robot.In_Position == TRUE){
					inst->Command.START     = FALSE;
					inst->Command.ID.Motion = MAIN_ID_EMPTY;

					inst->Internal.actual_state = ABBt_STATE_WAIT;
				}
			}
			break;
	}

	if(inst->Internal.actual_state == ABBt_STATE_MOVE_JOINT_CHECK || inst->Internal.actual_state == ABBt_STATE_MOVE_JOINT_EXECUTE ||
	inst->Internal.actual_state == ABBt_STATE_MOVE_TCP_CHECK || inst->Internal.actual_state == ABBt_STATE_MOVE_TCP_EXECUTE){
		if(inst->Command.STOP == TRUE){
			inst->Internal.actual_state = ABBt_STATE_STOP_EXECUTE;
		}
	}

	if(inst->Status.PLC.Module_OK == TRUE){
		inst->Status.PLC.Active = TRUE;

		Write_Data_PLC_to_ROB(inst);
	}else{
		inst->Status.PLC.Active = FALSE;
	}

	Update_Parameters(inst);
}

void Template_Reset(struct ABB_Library* inst){
	/**
	Description:
		Function to initialize and reset parameters of the template.

	Args:
		(1) inst [struct ABB_Library*]: Function block instance.
	*/

	/**
	 * INPUT VARIABLES
 	 */
	inst->Power_ON = inst->Power_OFF = FALSE;
	memset(&inst->Command, NULL, sizeof(inst->Command));
	memset(&inst->Parameter, NULL, sizeof(inst->Parameter));
	memset(&inst->Rob_Tool, NULL, sizeof(inst->Rob_Tool));

	/**
	 * OUTPUT VARIABLES
 	 */
	memset(&inst->Status, NULL, sizeof(inst->Status));
	memset(&inst->RT_Data, NULL, sizeof(inst->RT_Data));

	/**
	 * INTERNAL VARIABLES
 	 */
	inst->Internal.actual_state = inst->Internal.before_state = ABBt_STATE_INITIALIZATION;
	inst->Internal.Update.actual_state = UPT_STATE_INITIALIZATION;
}

void Update_Parameters(struct ABB_Library* inst){
	switch(inst->Internal.Update.actual_state){
		case UPT_STATE_INITIALIZATION:
			{
				if(inst->Status.Robot.Active == TRUE){
					inst->Internal.Update.actual_state = UPT_STATE_WAIT;
				}
			}
			break;

		case UPT_STATE_WAIT:
			{
				if(inst->Command.UPDATE == TRUE && inst->Command.ID.Update == UPT_ID_TRAJECTORY_JOINT){
					inst->Internal.Update.actual_state = UPT_STATE_JOINT_TRAJ_1;
				}else if(inst->Command.UPDATE == TRUE && inst->Command.ID.Update == UPT_ID_TRAJECTORY_TCP){
					inst->Internal.Update.actual_state = UPT_STATE_TCP_TRAJ_1;
				}else if(inst->Command.UPDATE == TRUE && inst->Command.ID.Update  == UPT_ID_ROB_TOOL){
					inst->Internal.Update.actual_state = UPT_STATE_RTOOL;
				}
			}
			break;

		case UPT_STATE_JOINT_TRAJ_1:
			{
				if(inst->Parameter.Trajectory_Size == inst->Internal.Update.ID){
					if(inst->Status.Robot.ID.Update == ABBu_STATE_INITIALIZATION){
						inst->Internal.Update.ID = NULL;
						aux_trajectory_ID                   = NULL;
						inst->Internal.Update.actual_state  = UPT_STATE_WAIT;
					}
				}else{
					if(inst->Status.Robot.ID.Update == ABBu_STATE_UPDATE_JOINT_TRAJ_3){
						aux_trajectory_ID = inst->Internal.Update.ID;

						inst->Command.UPDATE                = FALSE;
						inst->Command.ID.Update             = UPT_ID_EMPTY;
						inst->Internal.Update.actual_state  = UPT_STATE_JOINT_TRAJ_2;
					}
				}
			}
			break;

		case UPT_STATE_JOINT_TRAJ_2:
			{
				if(inst->Internal.Update.ID == aux_trajectory_ID){
					inst->Internal.Update.ID = aux_trajectory_ID + 1;
				}

				inst->Internal.Update.actual_state  = UPT_STATE_JOINT_TRAJ_3;
			}
			break;

		case UPT_STATE_JOINT_TRAJ_3:
			{
				inst->PROFINET_Mapping_OUT.SPEED = (unsigned char)inst->Parameter.Speed[inst->Internal.Update.ID - 1];
				inst->PROFINET_Mapping_OUT.ZONE  = (unsigned char)inst->Parameter.Zone[inst->Internal.Update.ID - 1];

				unsigned char i_j;
				for(i_j = 0; i_j < (unsigned char)(sizeof(inst->Parameter.Joint[0].Q)/sizeof(inst->Parameter.Joint[0].Q[0])); i_j++){
					if(inst->Parameter.Joint[inst->Internal.Update.ID - 1].Q[i_j] >= 0.0){
						inst->PROFINET_Mapping_OUT.JOINT_POS_SIGN.INPUT[i_j] = TRUE;
						inst->PROFINET_Mapping_OUT.JOINT_POS[i_j].INPUT      = (UINT)(ceil((inst->Parameter.Joint[inst->Internal.Update.ID - 1].Q[i_j] * inst->Internal.ACCURACY_FACTOR)*CEIL_DEFUALT_FACTOR)/CEIL_DEFUALT_FACTOR);
					}else{
						inst->PROFINET_Mapping_OUT.JOINT_POS_SIGN.INPUT[i_j] = FALSE;
						inst->PROFINET_Mapping_OUT.JOINT_POS[i_j].INPUT      = (-1) * ((UINT)(ceil((inst->Parameter.Joint[inst->Internal.Update.ID - 1].Q[i_j] * inst->Internal.ACCURACY_FACTOR)*CEIL_DEFUALT_FACTOR)/CEIL_DEFUALT_FACTOR));
					}

					Convert_UINT_To_USINT_Array(&inst->PROFINET_Mapping_OUT.JOINT_POS[i_j]);
				}

				Convert_BOOL_Array_To_USINT(&inst->PROFINET_Mapping_OUT.JOINT_POS_SIGN);

				inst->Status.PLC.Update_Done = TRUE;

				if(inst->Status.Robot.ID.Update == ABBu_STATE_UPDATE_JOINT_TRAJ_4){
					inst->Internal.Update.actual_state = UPT_STATE_JOINT_TRAJ_4;
				}
			}
			break;

		case UPT_STATE_JOINT_TRAJ_4:
			{
				inst->Status.PLC.Update_Done = FALSE;

				if(inst->Status.Robot.Update_Done == TRUE){
					inst->Internal.Update.actual_state = UPT_STATE_JOINT_TRAJ_1;
				}
			}
			break;

		case UPT_STATE_TCP_TRAJ_1:
			{
				if(inst->Parameter.Trajectory_Size == inst->Internal.Update.ID){
					if(inst->Status.Robot.ID.Update == ABBu_STATE_INITIALIZATION){
						inst->Internal.Update.ID = NULL;
						aux_trajectory_ID                   = NULL;
						inst->Internal.Update.actual_state  = UPT_STATE_WAIT;
					}
				}else{
					if(inst->Status.Robot.ID.Update == ABBu_STATE_UPDATE_TCP_TRAJ_3){
						aux_trajectory_ID = inst->Internal.Update.ID;

						inst->Command.UPDATE                = FALSE;
						inst->Command.ID.Update             = UPT_ID_EMPTY;
						inst->Internal.Update.actual_state  = UPT_STATE_TCP_TRAJ_2;
					}
				}
			}
			break;

		case UPT_STATE_TCP_TRAJ_2:
			{
				if(inst->Internal.Update.ID == aux_trajectory_ID){
					inst->Internal.Update.ID = aux_trajectory_ID + 1;
				}

				inst->Internal.Update.actual_state  = UPT_STATE_TCP_TRAJ_3;
			}
			break;

		case UPT_STATE_TCP_TRAJ_3:
			{
				inst->PROFINET_Mapping_OUT.SPEED = (unsigned char)inst->Parameter.Speed[inst->Internal.Update.ID - 1];
				inst->PROFINET_Mapping_OUT.ZONE  = (unsigned char)inst->Parameter.Zone[inst->Internal.Update.ID - 1];

				unsigned char i_tcp;
				for(i_tcp = 0; i_tcp < (unsigned char)(sizeof(inst->Parameter.TCP[0].Position)/sizeof(inst->Parameter.TCP[0].Position[0])); i_tcp++){
					if(inst->Parameter.TCP[inst->Internal.Update.ID - 1].Position[i_tcp] >= 0.0){
						inst->PROFINET_Mapping_OUT.TCP_SIGN.INPUT[i_tcp] = TRUE;
						inst->PROFINET_Mapping_OUT.TCP_POS[i_tcp].INPUT  = (UDINT)(ceil((inst->Parameter.TCP[inst->Internal.Update.ID - 1].Position[i_tcp] * inst->Internal.ACCURACY_FACTOR)*CEIL_DEFUALT_FACTOR)/CEIL_DEFUALT_FACTOR);
					}else{
						inst->PROFINET_Mapping_OUT.TCP_SIGN.INPUT[i_tcp] = FALSE;
						inst->PROFINET_Mapping_OUT.TCP_POS[i_tcp].INPUT  = (-1) * ((UDINT)(ceil((inst->Parameter.TCP[inst->Internal.Update.ID - 1].Position[i_tcp] * inst->Internal.ACCURACY_FACTOR)*CEIL_DEFUALT_FACTOR)/CEIL_DEFUALT_FACTOR));
					}
					Convert_UDINT_To_USINT_Array(&inst->PROFINET_Mapping_OUT.TCP_POS[i_tcp]);

					if(inst->Parameter.TCP[inst->Internal.Update.ID - 1].Rotation[i_tcp] >= 0.0){
						inst->PROFINET_Mapping_OUT.TCP_SIGN.INPUT[3 + i_tcp] = TRUE;
						inst->PROFINET_Mapping_OUT.TCP_ROT[i_tcp].INPUT  = (UDINT)(ceil((inst->Parameter.TCP[inst->Internal.Update.ID - 1].Rotation[i_tcp] * inst->Internal.ACCURACY_FACTOR)*CEIL_DEFUALT_FACTOR)/CEIL_DEFUALT_FACTOR);
					}else{
						inst->PROFINET_Mapping_OUT.TCP_SIGN.INPUT[3 + i_tcp] = FALSE;
						inst->PROFINET_Mapping_OUT.TCP_ROT[i_tcp].INPUT  = (-1) * ((UDINT)(ceil((inst->Parameter.TCP[inst->Internal.Update.ID - 1].Rotation[i_tcp] * inst->Internal.ACCURACY_FACTOR)*CEIL_DEFUALT_FACTOR)/CEIL_DEFUALT_FACTOR));
					}
					Convert_UINT_To_USINT_Array(&inst->PROFINET_Mapping_OUT.TCP_ROT[i_tcp]);
				}

				if(inst->Parameter.TCP[inst->Internal.Update.ID - 1].External_Position >= 0.0){
					inst->PROFINET_Mapping_OUT.TCP_SIGN.INPUT[6] = TRUE;
					inst->PROFINET_Mapping_OUT.TCP_EX_POS.INPUT  = (UDINT)(ceil((inst->Parameter.TCP[inst->Internal.Update.ID - 1].External_Position * inst->Internal.ACCURACY_FACTOR)*CEIL_DEFUALT_FACTOR)/CEIL_DEFUALT_FACTOR);
				}else{
					inst->PROFINET_Mapping_OUT.TCP_SIGN.INPUT[6] = FALSE;
					inst->PROFINET_Mapping_OUT.TCP_EX_POS.INPUT  = (-1) * ((UDINT)(ceil((inst->Parameter.TCP[inst->Internal.Update.ID - 1].External_Position * inst->Internal.ACCURACY_FACTOR)*CEIL_DEFUALT_FACTOR)/CEIL_DEFUALT_FACTOR));
				}

				Convert_BOOL_Array_To_USINT(&inst->PROFINET_Mapping_OUT.TCP_SIGN);

				unsigned char i_cfg;
				for(i_cfg = 0; i_cfg < (unsigned char)(sizeof(inst->Parameter.TCP[0].Configuration)/sizeof(inst->Parameter.TCP[0].Configuration[0])); i_cfg++){
					if(inst->Parameter.TCP[inst->Internal.Update.ID - 1].Configuration[i_cfg] >= 0){
						inst->PROFINET_Mapping_OUT.TCP_CFG_SIGN.INPUT[i_cfg] = TRUE;
						inst->PROFINET_Mapping_OUT.TCP_CFG[i_cfg]            = inst->Parameter.TCP[inst->Internal.Update.ID - 1].Configuration[i_cfg];
					}else{
						inst->PROFINET_Mapping_OUT.TCP_CFG_SIGN.INPUT[i_cfg] = FALSE;
						inst->PROFINET_Mapping_OUT.TCP_CFG[i_cfg]            = (-1) * inst->Parameter.TCP[inst->Internal.Update.ID - 1].Configuration[i_cfg];
					}
				}

				Convert_BOOL_Array_To_USINT(&inst->PROFINET_Mapping_OUT.TCP_CFG_SIGN);

				inst->Status.PLC.Update_Done = TRUE;

				if(inst->Status.Robot.ID.Update == ABBu_STATE_UPDATE_TCP_TRAJ_4){
					inst->Internal.Update.actual_state = UPT_STATE_TCP_TRAJ_4;
				}
			}
			break;

		case UPT_STATE_TCP_TRAJ_4:
			{
				inst->Status.PLC.Update_Done = FALSE;

				if(inst->Status.Robot.Update_Done == TRUE){
					inst->Internal.Update.actual_state = UPT_STATE_TCP_TRAJ_1;
				}
			}
			break;

		case UPT_STATE_RTOOL:
			{
				inst->PROFINET_Mapping_OUT.RTOOL_RH.INPUT[0] = inst->Rob_Tool.robHold;
				Convert_BOOL_Array_To_USINT(&inst->PROFINET_Mapping_OUT.RTOOL_RH);

				inst->PROFINET_Mapping_OUT.RTOOL_MASS.INPUT = (UINT)(ceil((inst->Rob_Tool.tLoad.mass * inst->Internal.ACCURACY_FACTOR)*CEIL_DEFUALT_FACTOR)/CEIL_DEFUALT_FACTOR);
				Convert_UINT_To_USINT_Array(&inst->PROFINET_Mapping_OUT.RTOOL_MASS);

				unsigned char i_tp;
				for(i_tp = 0; i_tp < (unsigned char)(sizeof(inst->Rob_Tool.tFrame.Position)/sizeof(inst->Rob_Tool.tFrame.Position[0])); i_tp++){
					if(inst->Rob_Tool.tFrame.Position[i_tp] >= 0.0){
						inst->PROFINET_Mapping_OUT.RTOOL_POS_SIGN.INPUT[i_tp] = TRUE;
						inst->PROFINET_Mapping_OUT.RTOOL_POS[i_tp].INPUT      = (UDINT)(ceil((inst->Rob_Tool.tFrame.Position[i_tp] * inst->Internal.ACCURACY_FACTOR)*CEIL_DEFUALT_FACTOR)/CEIL_DEFUALT_FACTOR);
					}else{
						inst->PROFINET_Mapping_OUT.RTOOL_POS_SIGN.INPUT[i_tp] = FALSE;
						inst->PROFINET_Mapping_OUT.RTOOL_POS[i_tp].INPUT      = (-1) * ((UDINT)(ceil((inst->Rob_Tool.tFrame.Position[i_tp] * inst->Internal.ACCURACY_FACTOR)*CEIL_DEFUALT_FACTOR)/CEIL_DEFUALT_FACTOR));
					}

					Convert_UINT_To_USINT_Array(&inst->PROFINET_Mapping_OUT.RTOOL_POS[i_tp]);

					if(inst->Rob_Tool.tLoad.center_of_gravity[i_tp] >= 0.0){
						inst->PROFINET_Mapping_OUT.RTOOL_COG_SIGN.INPUT[i_tp] = TRUE;
						inst->PROFINET_Mapping_OUT.RTOOL_COG[i_tp].INPUT      = (UDINT)(ceil((inst->Rob_Tool.tLoad.center_of_gravity[i_tp] * inst->Internal.ACCURACY_FACTOR)*CEIL_DEFUALT_FACTOR)/CEIL_DEFUALT_FACTOR);
					}else{
						inst->PROFINET_Mapping_OUT.RTOOL_COG_SIGN.INPUT[i_tp] = FALSE;
						inst->PROFINET_Mapping_OUT.RTOOL_COG[i_tp].INPUT      = (-1) * ((UDINT)(ceil((inst->Rob_Tool.tLoad.center_of_gravity[i_tp] * inst->Internal.ACCURACY_FACTOR)*CEIL_DEFUALT_FACTOR)/CEIL_DEFUALT_FACTOR));
					}

					Convert_UDINT_To_USINT_Array(&inst->PROFINET_Mapping_OUT.RTOOL_COG[i_tp]);

					inst->PROFINET_Mapping_OUT.RTOOL_MOI[i_tp].INPUT = (UDINT)(ceil((inst->Rob_Tool.tLoad.moment_of_inertia[i_tp] * inst->Internal.ACCURACY_FACTOR)*CEIL_DEFUALT_FACTOR)/CEIL_DEFUALT_FACTOR);
					Convert_UDINT_To_USINT_Array(&inst->PROFINET_Mapping_OUT.RTOOL_MOI[i_tp]);
				}

				Convert_BOOL_Array_To_USINT(&inst->PROFINET_Mapping_OUT.RTOOL_POS_SIGN);
				Convert_BOOL_Array_To_USINT(&inst->PROFINET_Mapping_OUT.RTOOL_COG_SIGN);

				unsigned char i_fp;
				for(i_fp = 0; i_fp < (unsigned char)(sizeof(inst->Rob_Tool.tFrame.Rotation)/sizeof(inst->Rob_Tool.tFrame.Rotation[0])); i_fp++){
					if(inst->Rob_Tool.tFrame.Rotation[i_fp] >= 0.0){
						inst->PROFINET_Mapping_OUT.RTOOL_ROT_QUAT_SIGN.INPUT[i_fp] = TRUE;
						inst->PROFINET_Mapping_OUT.RTOOL_ROT_QUAT[i_fp].INPUT      = (UDINT)(ceil((inst->Rob_Tool.tFrame.Rotation[i_fp] * inst->Internal.ACCURACY_FACTOR_QUATERNION)*CEIL_DEFUALT_FACTOR)/CEIL_DEFUALT_FACTOR);
					}else{
						inst->PROFINET_Mapping_OUT.RTOOL_ROT_QUAT_SIGN.INPUT[i_fp] = FALSE;
						inst->PROFINET_Mapping_OUT.RTOOL_ROT_QUAT[i_fp].INPUT      = (-1) * ((UDINT)(ceil((inst->Rob_Tool.tFrame.Rotation[i_fp] * inst->Internal.ACCURACY_FACTOR_QUATERNION)*CEIL_DEFUALT_FACTOR)/CEIL_DEFUALT_FACTOR));
					}

					Convert_UDINT_To_USINT_Array(&inst->PROFINET_Mapping_OUT.RTOOL_ROT_QUAT[i_fp]);

					if(inst->Rob_Tool.tLoad.intertial_axes[i_fp] >= 0.0){
						inst->PROFINET_Mapping_OUT.RTOOL_AOM_QUAT_SIGN.INPUT[i_fp] = TRUE;
						inst->PROFINET_Mapping_OUT.RTOOL_AOM_QUAT[i_fp].INPUT      = (UDINT)(ceil((inst->Rob_Tool.tLoad.intertial_axes[i_fp] * inst->Internal.ACCURACY_FACTOR_QUATERNION)*CEIL_DEFUALT_FACTOR)/CEIL_DEFUALT_FACTOR);
					}else{
						inst->PROFINET_Mapping_OUT.RTOOL_AOM_QUAT_SIGN.INPUT[i_fp] = FALSE;
						inst->PROFINET_Mapping_OUT.RTOOL_AOM_QUAT[i_fp].INPUT      = (-1) * ((UDINT)(ceil((inst->Rob_Tool.tLoad.intertial_axes[i_fp] * inst->Internal.ACCURACY_FACTOR_QUATERNION)*CEIL_DEFUALT_FACTOR)/CEIL_DEFUALT_FACTOR));
					}

					Convert_UDINT_To_USINT_Array(&inst->PROFINET_Mapping_OUT.RTOOL_AOM_QUAT[i_fp]);
				}

				Convert_BOOL_Array_To_USINT(&inst->PROFINET_Mapping_OUT.RTOOL_ROT_QUAT_SIGN);
				Convert_BOOL_Array_To_USINT(&inst->PROFINET_Mapping_OUT.RTOOL_AOM_QUAT_SIGN);

				if(inst->Status.Robot.Update_Done == TRUE){
					inst->Command.UPDATE    = FALSE;
					inst->Command.ID.Update = UPT_ID_EMPTY;

					inst->Internal.Update.actual_state = UPT_STATE_WAIT;
				}
			}
			break;
	}
}

void Write_Data_PLC_to_ROB(struct ABB_Library* inst){
	/**
	Description:
		Function to write the basic data to the robot controller.

	Args:
		(1) inst [struct ABB_Library*]: Function block instance.
	*/

	inst->PROFINET_Mapping_OUT.STATUS.INPUT[0] = inst->Status.PLC.Active;
	inst->PROFINET_Mapping_OUT.STATUS.INPUT[1] = inst->Status.PLC.Update_Done;
	Convert_BOOL_Array_To_USINT(&inst->PROFINET_Mapping_OUT.STATUS);

	inst->PROFINET_Mapping_OUT.SYSTEM.INPUT[0] = inst->Command.System.MOTOR_ON;
	inst->PROFINET_Mapping_OUT.SYSTEM.INPUT[1] = inst->Command.System.MOTOR_OFF;
	inst->PROFINET_Mapping_OUT.SYSTEM.INPUT[2] = inst->Command.System.PP_TO_MAIN;
	inst->PROFINET_Mapping_OUT.SYSTEM.INPUT[3] = inst->Command.System.START;
	inst->PROFINET_Mapping_OUT.SYSTEM.INPUT[4] = inst->Command.System.STOP;
	Convert_BOOL_Array_To_USINT(&inst->PROFINET_Mapping_OUT.SYSTEM);

	inst->PROFINET_Mapping_OUT.COMMAND_mID = inst->Command.ID.Motion;
	inst->PROFINET_Mapping_OUT.COMMAND_uID = inst->Command.ID.Update;

	inst->PROFINET_Mapping_OUT.COMMAND.INPUT[0] = inst->Command.START;
	inst->PROFINET_Mapping_OUT.COMMAND.INPUT[1] = inst->Command.STOP;
	inst->PROFINET_Mapping_OUT.COMMAND.INPUT[2] = inst->Command.UPDATE;
	Convert_BOOL_Array_To_USINT(&inst->PROFINET_Mapping_OUT.COMMAND);

	inst->PROFINET_Mapping_OUT.TRAJECTORY_SIZE.INPUT = inst->Parameter.Trajectory_Size;
	Convert_UINT_To_USINT_Array(&inst->PROFINET_Mapping_OUT.TRAJECTORY_SIZE);
}

void Read_Data_ROB_to_PLC(struct ABB_Library* inst){
	/**
	Description:
		Function to collect data from the robot controller.

	Args:
		(1) inst [struct ABB_Library*]: Function block instance.
	*/

	Convert_USINT_To_BOOL_Array(&inst->PROFINET_Mapping_IN.STATUS);
	inst->Status.Robot.Active      = inst->PROFINET_Mapping_IN.STATUS.OUTPUT[0];
	inst->Status.Robot.Update_Done = inst->PROFINET_Mapping_IN.STATUS.OUTPUT[1];
	inst->Status.Robot.In_Position = inst->PROFINET_Mapping_IN.STATUS.OUTPUT[2];

	inst->Status.Robot.ID.Motion = inst->PROFINET_Mapping_IN.STATE_mID;

	Convert_USINT_To_BOOL_Array(&inst->PROFINET_Mapping_IN.SYSTEM);
	inst->Status.Robot.System.MOTOR_ON  = inst->PROFINET_Mapping_IN.SYSTEM.OUTPUT[0];
	inst->Status.Robot.System.MOTOR_OFF = inst->PROFINET_Mapping_IN.SYSTEM.OUTPUT[1];
	inst->Status.Robot.System.PP_MOVED  = inst->PROFINET_Mapping_IN.SYSTEM.OUTPUT[2];
	inst->Status.Robot.System.CYCLE_ON  = inst->PROFINET_Mapping_IN.SYSTEM.OUTPUT[3];

	inst->Status.Robot.ID.Update = inst->PROFINET_Mapping_IN.STATE_uID;

	Convert_USINT_Array_To_UINT(&inst->PROFINET_Mapping_IN.MOTION_TRAJECTORY_ID);
	inst->Status.Robot.Trajectory_ID = inst->PROFINET_Mapping_IN.MOTION_TRAJECTORY_ID.OUTPUT;

	Convert_USINT_To_BOOL_Array(&inst->PROFINET_Mapping_IN.JOINT_POS_SIGN);
	unsigned char i_j;
	for(i_j = 0; i_j < (unsigned char)(sizeof(inst->RT_Data.Q)/sizeof(inst->RT_Data.Q[0])); i_j++){
		Convert_USINT_Array_To_UINT(&inst->PROFINET_Mapping_IN.JOINT_POS[i_j]);

		if(inst->PROFINET_Mapping_IN.JOINT_POS_SIGN.OUTPUT[i_j] == TRUE){
			inst->RT_Data.Q[i_j] = (REAL)(inst->PROFINET_Mapping_IN.JOINT_POS[i_j].OUTPUT) / inst->Internal.ACCURACY_FACTOR;
		}else{
			inst->RT_Data.Q[i_j] = (-1) * ((REAL)(inst->PROFINET_Mapping_IN.JOINT_POS[i_j].OUTPUT) / inst->Internal.ACCURACY_FACTOR);
		}
	}

	Convert_USINT_To_BOOL_Array(&inst->PROFINET_Mapping_IN.TCP_SIGN);
	unsigned char i_tcp;
	for(i_tcp = 0; i_tcp < (unsigned char)(sizeof(inst->RT_Data.TCP.Position)/sizeof(inst->RT_Data.TCP.Position[0])); i_tcp++){
		Convert_USINT_Array_To_UDINT(&inst->PROFINET_Mapping_IN.TCP_POS[i_tcp]);
		if(inst->PROFINET_Mapping_IN.TCP_SIGN.OUTPUT[i_tcp] == TRUE){
			inst->RT_Data.TCP.Position[i_tcp] = (REAL)(inst->PROFINET_Mapping_IN.TCP_POS[i_tcp].OUTPUT) / inst->Internal.ACCURACY_FACTOR;
		}else{
			inst->RT_Data.TCP.Position[i_tcp] = (-1) * ((REAL)(inst->PROFINET_Mapping_IN.TCP_POS[i_tcp].OUTPUT) / inst->Internal.ACCURACY_FACTOR);
		}

		Convert_USINT_Array_To_UINT(&inst->PROFINET_Mapping_IN.TCP_ROT[i_tcp]);
		if(inst->PROFINET_Mapping_IN.TCP_SIGN.OUTPUT[i_tcp + 3] == TRUE){
			inst->RT_Data.TCP.Rotation[i_tcp] = (REAL)(inst->PROFINET_Mapping_IN.TCP_ROT[i_tcp].OUTPUT) / inst->Internal.ACCURACY_FACTOR;
		}else{
			inst->RT_Data.TCP.Rotation[i_tcp] = (-1) * ((REAL)(inst->PROFINET_Mapping_IN.TCP_ROT[i_tcp].OUTPUT) / inst->Internal.ACCURACY_FACTOR);
		}
	}

	Convert_USINT_Array_To_UINT(&inst->PROFINET_Mapping_IN.TCP_EX_POS);
	if(inst->PROFINET_Mapping_IN.TCP_SIGN.OUTPUT[6] == TRUE){
		inst->RT_Data.TCP.External_Position = (REAL)(inst->PROFINET_Mapping_IN.TCP_EX_POS.OUTPUT) / inst->Internal.ACCURACY_FACTOR;
	}else{
		inst->RT_Data.TCP.External_Position = (-1) * ((REAL)(inst->PROFINET_Mapping_IN.TCP_EX_POS.OUTPUT) / inst->Internal.ACCURACY_FACTOR);
	}

	Convert_USINT_To_BOOL_Array(&inst->PROFINET_Mapping_IN.TCP_CFG_SIGN);
	unsigned char i_cfg;
	for(i_cfg = 0; i_cfg < (unsigned char)(sizeof(inst->RT_Data.TCP.Configuration)/sizeof(inst->RT_Data.TCP.Configuration[0])); i_cfg++){
		if(inst->PROFINET_Mapping_IN.TCP_CFG_SIGN.OUTPUT[i_cfg] == TRUE){
			inst->RT_Data.TCP.Configuration[i_cfg] = (SINT)inst->PROFINET_Mapping_IN.TCP_CFG[i_cfg];
		}else{
			inst->RT_Data.TCP.Configuration[i_cfg] = (SINT)((-1) * inst->PROFINET_Mapping_IN.TCP_CFG[i_cfg]);
		}
	}
}

#endif
```

#### Types.typ - not listed in the package file held
```iecst
TYPE
	Traj_Str : 	STRUCT
		Targets : Targets_Str;
		Length : USINT;
		Iteration : USINT;
	END_STRUCT;
	Targets_Str : 	STRUCT
		Position : ARRAY[0..99]OF Targets_Position_Str;
		Speed : ARRAY[0..99]OF USINT;
		Zone : ARRAY[0..99]OF USINT;
	END_STRUCT;
	Targets_Position_Str : 	STRUCT
		Q : ARRAY[0..5]OF REAL;
		Q_Ex : ARRAY[0..5]OF REAL;
	END_STRUCT;
END_TYPE
```

- Visualisation Logical/mappView (not shown)

### Program Logical/axCtrl_T (ANSIC)

#### ax_ctrl.c - Init, cyclic, exit code
```c
/**

 * MIT License

 * Copyright(c) 2020 Roman Parak
 * Permission is hereby granted, free of charge, to any person obtaining a copy
 * of this software and associated documentation files (the "Software"), to deal
 * in the Software without restriction, including without limitation the rights
 * to use, copy, modify, merge, publish, distribute, sublicense, and/or sell
 * copies of the Software, and to permit persons to whom the Software is
 * furnished to do so, subject to the following conditions:
 * The above copyright notice and this permission notice shall be included in all
 * copies or substantial portions of the Software.
 * THE SOFTWARE IS PROVIDED "AS IS", WITHOUT WARRANTY OF ANY KIND, EXPRESS OR
 * IMPLIED, INCLUDING BUT NOT LIMITED TO THE WARRANTIES OF MERCHANTABILITY,
 * FITNESS FOR A PARTICULAR PURPOSE AND NONINFRINGEMENT. IN NO EVENT SHALL THE
 * AUTHORS OR COPYRIGHT HOLDERS BE LIABLE FOR ANY CLAIM, DAMAGES OR OTHER
 * LIABILITY, WHETHER IN AN ACTION OF CONTRACT, TORT OR OTHERWISE, ARISING FROM,
 * OUT OF OR IN CONNECTION WITH THE SOFTWARE OR THE USE OR OTHER DEALINGS IN THE
 * SOFTWARE.
 */

/**
 * Author   : Roman Parak
 * Email    : Roman.Parak@outlook.com
 * Date     : 12.12.2020
 * File Name: axCtrl_T.c
 */

/** < Include B&R Automation libraries (declarations for B&R ANSI C extensions) */
#include <bur/plctypes.h>

#ifdef _DEFAULT_INCLUDES
#include <AsDefault.h>
#endif

/** < Include header file with specified structures / enums, etc. */
#include "ax_ctrl.h"

/// Function block for controlling all basic functions of a single axis
_LOCAL struct MpAxisBasic MpAxisBasic_0;
/// Standard parameters for controlling axes (position, velocity, etc.)
_LOCAL struct MpAxisBasicParType AxisParameters;

/// Custom structure for axis control and data collection (more in the header file -> axCtrl_T.h)
_LOCAL struct motion_ctrl_main ctrl_lin_ax_0;

/**
 * Program Intitialization
 */
void _INIT ProgramInit(void)
{
	/// Declaration of function block inputs
	MpAxisBasic_0.Enable     = 1;			    ///< Enables the function block
	MpAxisBasic_0.MpLink     = &gAxis_Mech_01;		///< Connection to mapp (MpLink of an MpAxisBasic configuration)
	MpAxisBasic_0.Parameters = &AxisParameters;	///< Function block parameters

	/// Set initialization state to default
	ctrl_lin_ax_0.actual_state = LIN_AX_CTRL_ACTIVE;
}

/**
 * Program Cyclic
 *
 * Duration (Cycle Time): 1000 [µs]
 * Tolerance            : 0    [µs]
 */
void _CYCLIC ProgramCyclic(void)
{
	/**
	 * Main state machine for control of a single axis.
	 *
	 * Number of states: 8 (for more information -> axCtrl_T.h)
	 */
	switch(ctrl_lin_ax_0.actual_state){
		case LIN_AX_CTRL_ACTIVE: ///< The Function block is active.
			{
				if(ctrl_lin_ax_0.read.is_active == 1){
					ctrl_lin_ax_0.actual_state = LIN_AX_CTRL_POWER;
				}
			}
			break;
		case LIN_AX_CTRL_POWER: ///< Axis is power on.
			{
				if(ctrl_lin_ax_0.read.power_on == 1){
					ctrl_lin_ax_0.actual_state = LIN_AX_CTRL_HOME;
				}
			}
			break;
		case LIN_AX_CTRL_HOME: ///< Axis is homed.
			{
				if(ctrl_lin_ax_0.read.is_homed == 1){
					MpAxisBasic_0.Home = 0;
					ctrl_lin_ax_0.actual_state = LIN_AX_CTRL_WAIT;
				}
			}
			break;
		case LIN_AX_CTRL_WAIT: ///< Wait for the command.
			{
				GLOBAL_POS = MpAxisBasic_0.Position;
				GLOBAL_START = 1;

				if(ctrl_lin_ax_0.cmd.move_absolute_postion == 1){
					ctrl_lin_ax_0.actual_state = LIN_AX_CTRL_MOVE_1;
				}
			}
			break;
		case LIN_AX_CTRL_MOVE_1: ///< Move Axis (1) -> Set Parameters.
			{
				ctrl_lin_ax_0.cmd.move_absolute_postion = 0;

				AxisParameters.Position     = ctrl_lin_ax_0.write.position;
				AxisParameters.Velocity     = ctrl_lin_ax_0.write.velocity;
				AxisParameters.Acceleration = ctrl_lin_ax_0.write.acceleration;
				AxisParameters.Deceleration = ctrl_lin_ax_0.write.deceleration;

				ctrl_lin_ax_0.read.set_position = ctrl_lin_ax_0.write.position;

				/**
				 * Check the direction of movement of the axis from the actual position.
				 *
				 * Set Position >= Actual Position -> Velocity (+)
				 * Set Position < Actual Position  -> Velocity (-)
				 */
				if(ctrl_lin_ax_0.read.set_position >= ctrl_lin_ax_0.read.actual_position){
					ctrl_lin_ax_0.read.set_velocity = ctrl_lin_ax_0.write.velocity;
				}else if(ctrl_lin_ax_0.read.set_position < ctrl_lin_ax_0.read.actual_position){
					ctrl_lin_ax_0.read.set_velocity = (-1)*ctrl_lin_ax_0.write.velocity;
				}

				MpAxisBasic_0.MoveAbsolute = 1;

				if(MpAxisBasic_0.MoveActive == 1){
					ctrl_lin_ax_0.actual_state = LIN_AX_CTRL_MOVE_2;
				}
			}
			break;
		case LIN_AX_CTRL_MOVE_2: ///< Move Axis (2) -> Wait until the axis is in specified position.
			{
				if(MpAxisBasic_0.InPosition == 1 && MpAxisBasic_0.MoveDone == 1){
					ctrl_lin_ax_0.read.set_velocity = 0.0;
					MpAxisBasic_0.MoveAbsolute = 0;
					ctrl_lin_ax_0.actual_state = LIN_AX_CTRL_WAIT;
				}
			}
			break;
		case LIN_AX_CTRL_ERROR: ///< The function block is in an error state, wait for reset.
			{
				MpAxisBasic_0.MoveAbsolute = 0;

				ctrl_lin_ax_0.write.position     = 0.0;
				ctrl_lin_ax_0.write.velocity     = 0.0;
				ctrl_lin_ax_0.write.acceleration = 0.0;
				ctrl_lin_ax_0.write.deceleration = 0.0;

				if(ctrl_lin_ax_0.read.error == 0){
					ctrl_lin_ax_0.actual_state = LIN_AX_CTRL_WAIT;
				}
			}
			break;
	}

	/// write inputs to the function block
	MpAxisBasic_0.Power      = ctrl_lin_ax_0.cmd.power;
	MpAxisBasic_0.Home       = ctrl_lin_ax_0.cmd.home;
	MpAxisBasic_0.ErrorReset = ctrl_lin_ax_0.cmd.reset_error;

	/// call MpAxisBasic function block
	MpAxisBasic(&MpAxisBasic_0);

	GLOBAL_VEL = MpAxisBasic_0.Velocity;

	/// read outputs from the function block
	ctrl_lin_ax_0.read.is_active        = MpAxisBasic_0.Active;
	ctrl_lin_ax_0.read.power_on         = MpAxisBasic_0.PowerOn;
	ctrl_lin_ax_0.read.is_homed         = MpAxisBasic_0.IsHomed;
	ctrl_lin_ax_0.read.error            = MpAxisBasic_0.Error;
	ctrl_lin_ax_0.read.actual_position  = MpAxisBasic_0.Position;
	ctrl_lin_ax_0.read.actual_velocity  = MpAxisBasic_0.Velocity;

	/**
	 * Digital twin (scene viewer) -> reading the actual position and
	 * transforming the specified axis units into millimeters.
	 */
	ctrl_lin_ax_0.write.dT.position = MpAxisBasic_0.Position;
	/**
	 * Error detection (cyclic reading in time).
	 *
	 * After detecting one or more errors, change the state on the main
	 * state machine and wait for the error reset command.
	 */
	if(ctrl_lin_ax_0.read.error == 1){
		ctrl_lin_ax_0.actual_state = LIN_AX_CTRL_ERROR;
	}

}
```

### Program Logical/axStream_T

#### Main.c
```c
#include <bur/plctypes.h>

#ifdef _DEFAULT_INCLUDES
#include <AsDefault.h>
#endif

/// Function block for controlling all basic functions of a single axis
_LOCAL struct MpAxisBasic MpAxisBasic_0;
_LOCAL struct MpAxisCyclicSet MpAxisCyclicSet_0;
/// Standard parameters for controlling axes (position, velocity, etc.)
_LOCAL struct MpAxisBasicParType AxisParameters;
_LOCAL struct MpAxisCyclicSetParType AxisCyclicParameters;

_LOCAL USINT actual_state;
_LOCAL LREAL dt_position;

// add start/stop of the streaming!!!

void _INIT ProgramInit(void)
{
	/// Declaration of function block inputs
	MpAxisBasic_0.Enable     = 1;			    ///< Enables the function block
	MpAxisBasic_0.MpLink     = &gAxis_Mech_02;		///< Connection to mapp (MpLink of an MpAxisBasic configuration)
	MpAxisBasic_0.Parameters = &AxisParameters;	///< Function block parameters
	// ...
	AxisParameters.Velocity     = 500;
	AxisParameters.Acceleration = 2000;
	AxisParameters.Deceleration = 2000;

	MpAxisCyclicSet_0.Enable = 1;
	MpAxisCyclicSet_0.MpLink = &gAxis_Mech_02;
	MpAxisCyclicSet_0.Parameters = &AxisCyclicParameters;
	AxisCyclicParameters.MoveCyclicVelocity.Mode = mcAXIS_MCV_MODE_MOVE_CYC_VEL;
	AxisCyclicParameters.MoveCyclicVelocity.InterpolationMode = mcIPLM_DEFAULT;
	AxisCyclicParameters.MoveCyclicVelocity.Acceleration = 20000;
	AxisCyclicParameters.MoveCyclicVelocity.Deceleration = 20000;

	actual_state = 0;
}

void _CYCLIC ProgramCyclic(void)
{
	switch(actual_state){
		case 0:
			{
				if(MpAxisBasic_0.Active == 1 && GLOBAL_START == 1){
					actual_state = 1;
				}
			}
			break;
		case 1:
			{
				MpAxisBasic_0.Power = 1;

				if(MpAxisBasic_0.PowerOn == 1){
					actual_state = 2;

				}
			}
			break;
		case 2:
			{
				MpAxisBasic_0.Home = 1;

				if(MpAxisBasic_0.IsHomed == 1){
					MpAxisBasic_0.Home = 0;
					actual_state = 6;

				}
			}
			break;

		case 6:
			{
				MpAxisCyclicSet_0.MoveCyclicVelocity = 1;

				if(MpAxisCyclicSet_0.MoveCyclicVelocityActive == 1){
					actual_state = 7;
				}
			}
			break;

		case 7:
			{
				MpAxisCyclicSet_0.CyclicVelocity = GLOBAL_VEL;
			}
			break;

	}

	/// call MpAxisBasic function block
	MpAxisBasic(&MpAxisBasic_0);
	MpAxisCyclicSet(&MpAxisCyclicSet_0);

	dt_position = MpAxisBasic_0.Position;
}
```

### Program Logical/T_MECH_ID_1

#### Main.c
```c
#include <bur/plctypes.h>

#ifdef _DEFAULT_INCLUDES
#include <AsDefault.h>
#endif

#include "Main.h"

_LOCAL struct MpAxisBasic MpAxisBasic_0;
_LOCAL struct MpAxisBasicParType AxisParameters;
_LOCAL enum Mechanism_State_ID_enum state_id;

void _INIT ProgramInit(void)
{
	MpAxisBasic_0.Enable     = 1;
	MpAxisBasic_0.MpLink     = &gAxis_Mech_01;
	MpAxisBasic_0.Parameters = &AxisParameters;

	Trajectory_Str.Targets.Position[0] = 100.0;
	Trajectory_Str.Targets.Position[1] = 1100.0;
	Trajectory_Str.Targets.Position[2] = 700.0;
	Trajectory_Str.Targets.Position[3] = 300.0;
	Trajectory_Str.Targets.Position[4] = 1200.0;

	Trajectory_Str.Targets.Velocity[0] = 500.0;
	Trajectory_Str.Targets.Velocity[1] = 1000.0;
	Trajectory_Str.Targets.Velocity[2] = 200.0;
	Trajectory_Str.Targets.Velocity[3] = 1500.0;
	Trajectory_Str.Targets.Velocity[4] = 400.0;

	Trajectory_Str.Length = 5;

	state_id = STATE_ID_ACTIVE;
}

void _CYCLIC ProgramCyclic(void)
{
	switch(state_id){
		case STATE_ID_ACTIVE:
			{
				if(Global_MappView_Str.Mech_Id_1.Info.Active == 1){
					state_id = STATE_ID_POWER;
				}
			}
			break;

		case STATE_ID_POWER:
			{
				if(Global_MappView_Str.Mech_Id_1.Info.Power == 1){
					state_id = STATE_ID_HOME;
				}
			}
			break;

		case STATE_ID_HOME:
			{
				if(Global_MappView_Str.Mech_Id_1.Info.Home == 1){
					MpAxisBasic_0.Home = 0;
					Global_MappView_Str.Mech_Id_1.Command.Home = 0;
					state_id = STATE_ID_WAIT;
				}
			}
			break;

		case STATE_ID_WAIT:
			{
				if(Global_MappView_Str.Mech_Id_1.Command.Home == 1){
					state_id = STATE_ID_HOME_UPDATE_PARAMETERS;
				}

				if(Global_MappView_Str.Mech_Id_1.Command.Start == 1){
					Trajectory_Str.Iteration = 0;
					state_id = STATE_ID_UPDATE_PARAMETERS;
				}
			}
			break;

		case STATE_ID_UPDATE_PARAMETERS:
			{
				AxisParameters.Position     = Trajectory_Str.Targets.Position[Trajectory_Str.Iteration];
				AxisParameters.Velocity     = Trajectory_Str.Targets.Velocity[Trajectory_Str.Iteration];
				AxisParameters.Acceleration = Trajectory_Str.Targets.Velocity[Trajectory_Str.Iteration]*10;
				AxisParameters.Deceleration = AxisParameters.Acceleration;

				MpAxisBasic_0.Update = 1;
				if(MpAxisBasic_0.UpdateDone == 1){
					state_id = STATE_ID_MOTION_1;
				}
			}
			break;

		case STATE_ID_MOTION_1:
			{
				MpAxisBasic_0.MoveAbsolute = 1;
				if(MpAxisBasic_0.MoveActive == 1){
					state_id = STATE_ID_MOTION_2;
				}
			}
			break;

		case STATE_ID_MOTION_2:
			{
				if(Global_MappView_Str.Mech_Id_1.Command.Stop == 1){
					state_id = STATE_ID_STOP;
				}else{
					if(MpAxisBasic_0.InPosition == 1 && MpAxisBasic_0.MoveDone == 1){
						MpAxisBasic_0.MoveAbsolute = 0;

						if(Trajectory_Str.Iteration == Trajectory_Str.Length - 1){
							state_id = STATE_ID_WAIT;
						}else{
							Trajectory_Str.Iteration++;
							state_id = STATE_ID_UPDATE_PARAMETERS;
						}
					}
				}
			}
			break;

		case STATE_ID_HOME_UPDATE_PARAMETERS:
			{
				AxisParameters.Position     = 700.0;
				AxisParameters.Velocity     = 500.0;
				AxisParameters.Acceleration = 5000.0;
				AxisParameters.Deceleration = 5000.0;

				MpAxisBasic_0.Update = 1;
				if(MpAxisBasic_0.UpdateDone == 1){
					state_id = STATE_ID_HOME_MOTION_1;
				}
			}
			break;

		case STATE_ID_HOME_MOTION_1:
			{
				MpAxisBasic_0.MoveAbsolute = 1;
				if(MpAxisBasic_0.MoveActive == 1){
					state_id = STATE_ID_HOME_MOTION_2;
				}
			}
			break;

		case STATE_ID_HOME_MOTION_2:
			{
				if(MpAxisBasic_0.InPosition == 1 && MpAxisBasic_0.MoveDone == 1){
					MpAxisBasic_0.MoveAbsolute = 0;
					Global_MappView_Str.Mech_Id_1.Command.Home = 0;
					state_id = STATE_ID_WAIT;
				}
			}
			break;

		case STATE_ID_STOP:
			{
				Global_MappView_Str.Mech_Id_1.Command.Stop  = 0;
				Global_MappView_Str.Mech_Id_1.Command.Start = 0;

				MpAxisBasic_0.MoveAbsolute = 0;
				if(MpAxisBasic_0.MoveActive == 0){
					state_id = STATE_ID_WAIT;
				}
			}
			break;

		case STATE_ID_SAFETY:
			{
			}
			break;

		case STATE_ID_ERROR:
			{
				if(Global_MappView_Str.Mech_Id_1.Info.Error == 1){
					state_id = STATE_ID_WAIT;
				}
			}
			break;

	}

	MpAxisBasic_0.Power      = Global_MappView_Str.Mech_Id_1.Command.Power;
	if(Global_MappView_Str.Mech_Id_1.Command.Home == 1 && Global_MappView_Str.Mech_Id_1.Info.Home == 0){
		MpAxisBasic_0.Home = 1;
	}
	MpAxisBasic_0.ErrorReset = Global_MappView_Str.Mech_Id_1.Command.Reset_Error;

	MpAxisBasic(&MpAxisBasic_0);

	Global_MappView_Str.Mech_Id_1.Info.Active = MpAxisBasic_0.Active;
	Global_MappView_Str.Mech_Id_1.Info.Power  = MpAxisBasic_0.PowerOn;
	Global_MappView_Str.Mech_Id_1.Info.Home   = MpAxisBasic_0.IsHomed;
	Global_MappView_Str.Mech_Id_1.Info.Error  = MpAxisBasic_0.Error;
	Global_MappView_Str.Mech_Id_1.Position = MpAxisBasic_0.Position;

	if(Global_MappView_Str.Mech_Id_1.Info.Error == 1){
		state_id = STATE_ID_ERROR;
	}

}
```

### Program Logical/T_MECH_ID_2

#### Main.h
```c
#include <bur/plctypes.h>

#ifdef _DEFAULT_INCLUDES
	#include <AsDefault.h>
#endif

typedef enum Mechanism_State_ID_enum{
	STATE_ID_ACTIVE,
	STATE_ID_POWER,
	STATE_ID_HOME,
	STATE_ID_WAIT,
	STATE_ID_UPDATE_PARAMETERS,
	STATE_ID_MOTION_1,
	STATE_ID_MOTION_2,
	STATE_ID_HOME_UPDATE_PARAMETERS,
	STATE_ID_HOME_MOTION_1,
	STATE_ID_HOME_MOTION_2,
	STATE_ID_STOP,
	STATE_ID_SAFETY,
	STATE_ID_ERROR
}Mechanism_State_ID_enum;
```

#### Main.c
```c
#include <bur/plctypes.h>

#ifdef _DEFAULT_INCLUDES
#include <AsDefault.h>
#endif

#include "Main.h"

_LOCAL struct MpAxisBasic MpAxisBasic_0;
_LOCAL struct MpAxisBasicParType AxisParameters;
_LOCAL enum Mechanism_State_ID_enum state_id;

void _INIT ProgramInit(void)
{
	MpAxisBasic_0.Enable     = 1;
	MpAxisBasic_0.MpLink     = &gAxis_Mech_02;
	MpAxisBasic_0.Parameters = &AxisParameters;

	Trajectory_Str.Targets.Position[0] = 1100.0;
	Trajectory_Str.Targets.Position[1] = 100.0;
	Trajectory_Str.Targets.Position[2] = 700.0;
	Trajectory_Str.Targets.Position[3] = 1200.0;
	Trajectory_Str.Targets.Position[4] = 300.0;

	Trajectory_Str.Targets.Velocity[0] = 500.0;
	Trajectory_Str.Targets.Velocity[1] = 1000.0;
	Trajectory_Str.Targets.Velocity[2] = 200.0;
	Trajectory_Str.Targets.Velocity[3] = 1500.0;
	Trajectory_Str.Targets.Velocity[4] = 400.0;

	Trajectory_Str.Length = 5;

	state_id = STATE_ID_ACTIVE;
}

void _CYCLIC ProgramCyclic(void)
{
	switch(state_id){
		case STATE_ID_ACTIVE:
			{
				if(Global_MappView_Str.Mech_Id_2.Info.Active == 1){
					state_id = STATE_ID_POWER;
				}
			}
			break;

		case STATE_ID_POWER:
			{
				if(Global_MappView_Str.Mech_Id_2.Info.Power == 1){
					state_id = STATE_ID_HOME;
				}
			}
			break;

		case STATE_ID_HOME:
			{
				if(Global_MappView_Str.Mech_Id_2.Info.Home == 1){
					MpAxisBasic_0.Home = 0;
					Global_MappView_Str.Mech_Id_2.Command.Home = 0;
					state_id = STATE_ID_WAIT;
				}
			}
			break;

		case STATE_ID_WAIT:
			{
				if(Global_MappView_Str.Mech_Id_2.Command.Home == 1){
					state_id = STATE_ID_HOME_UPDATE_PARAMETERS;
				}

				if(Global_MappView_Str.Mech_Id_2.Command.Start == 1){
					Trajectory_Str.Iteration = 0;
					state_id = STATE_ID_UPDATE_PARAMETERS;
				}
			}
			break;

		case STATE_ID_UPDATE_PARAMETERS:
			{
				AxisParameters.Position     = Trajectory_Str.Targets.Position[Trajectory_Str.Iteration];
				AxisParameters.Velocity     = Trajectory_Str.Targets.Velocity[Trajectory_Str.Iteration];
				AxisParameters.Acceleration = Trajectory_Str.Targets.Velocity[Trajectory_Str.Iteration]*10;
				AxisParameters.Deceleration = AxisParameters.Acceleration;

				MpAxisBasic_0.Update = 1;
				if(MpAxisBasic_0.UpdateDone == 1){
					state_id = STATE_ID_MOTION_1;
				}
			}
			break;

		case STATE_ID_MOTION_1:
			{
				MpAxisBasic_0.MoveAbsolute = 1;
				if(MpAxisBasic_0.MoveActive == 1){
					state_id = STATE_ID_MOTION_2;
				}
			}
			break;

		case STATE_ID_MOTION_2:
			{
				if(Global_MappView_Str.Mech_Id_2.Command.Stop == 1){
					state_id = STATE_ID_STOP;
				}else{
					if(MpAxisBasic_0.InPosition == 1 && MpAxisBasic_0.MoveDone == 1){
						MpAxisBasic_0.MoveAbsolute = 0;

						if(Trajectory_Str.Iteration == Trajectory_Str.Length - 1){
							state_id = STATE_ID_WAIT;
						}else{
							Trajectory_Str.Iteration++;
							state_id = STATE_ID_UPDATE_PARAMETERS;
						}
					}
				}
			}
			break;

		case STATE_ID_HOME_UPDATE_PARAMETERS:
			{
				AxisParameters.Position     = 700.0;
				AxisParameters.Velocity     = 500.0;
				AxisParameters.Acceleration = 5000.0;
				AxisParameters.Deceleration = 5000.0;

				MpAxisBasic_0.Update = 1;
				if(MpAxisBasic_0.UpdateDone == 1){
					state_id = STATE_ID_HOME_MOTION_1;
				}
			}
			break;

		case STATE_ID_HOME_MOTION_1:
			{
				MpAxisBasic_0.MoveAbsolute = 1;
				if(MpAxisBasic_0.MoveActive == 1){
					state_id = STATE_ID_HOME_MOTION_2;
				}
			}
			break;

		case STATE_ID_HOME_MOTION_2:
			{
				if(MpAxisBasic_0.InPosition == 1 && MpAxisBasic_0.MoveDone == 1){
					MpAxisBasic_0.MoveAbsolute = 0;
					Global_MappView_Str.Mech_Id_2.Command.Home = 0;
					state_id = STATE_ID_WAIT;
				}
			}
			break;

		case STATE_ID_STOP:
			{
				Global_MappView_Str.Mech_Id_2.Command.Stop  = 0;
				Global_MappView_Str.Mech_Id_2.Command.Start = 0;

				MpAxisBasic_0.MoveAbsolute = 0;
				if(MpAxisBasic_0.MoveActive == 0){
					state_id = STATE_ID_WAIT;
				}
			}
			break;

		case STATE_ID_SAFETY:
			{
			}
			break;

		case STATE_ID_ERROR:
			{
				if(Global_MappView_Str.Mech_Id_2.Info.Error == 1){
					state_id = STATE_ID_WAIT;
				}
			}
			break;

	}

	MpAxisBasic_0.Power      = Global_MappView_Str.Mech_Id_2.Command.Power;
	if(Global_MappView_Str.Mech_Id_2.Command.Home == 1 && Global_MappView_Str.Mech_Id_2.Info.Home == 0){
		MpAxisBasic_0.Home = 1;
	}
	MpAxisBasic_0.ErrorReset = Global_MappView_Str.Mech_Id_2.Command.Reset_Error;

	MpAxisBasic(&MpAxisBasic_0);

	Global_MappView_Str.Mech_Id_2.Info.Active = MpAxisBasic_0.Active;
	Global_MappView_Str.Mech_Id_2.Info.Power  = MpAxisBasic_0.PowerOn;
	Global_MappView_Str.Mech_Id_2.Info.Home   = MpAxisBasic_0.IsHomed;
	Global_MappView_Str.Mech_Id_2.Info.Error  = MpAxisBasic_0.Error;
	Global_MappView_Str.Mech_Id_2.Position = MpAxisBasic_0.Position;

	if(Global_MappView_Str.Mech_Id_2.Info.Error == 1){
		state_id = STATE_ID_ERROR;
	}
}
```

### Program Logical/T_MECH_ID_3

#### Types.typ
```iecst
TYPE
	Traj_Str : 	STRUCT
		Targets : Targets_Str;
		Length : USINT;
		Iteration : USINT;
	END_STRUCT;
	Targets_Str : 	STRUCT
		Position : ARRAY[0..100]OF LREAL;
		Velocity : ARRAY[0..100]OF REAL;
	END_STRUCT;
END_TYPE
```

#### Main.c
```c
#include <bur/plctypes.h>

#ifdef _DEFAULT_INCLUDES
#include <AsDefault.h>
#endif

#include "Main.h"

_LOCAL struct MpAxisBasic MpAxisBasic_0;
_LOCAL struct MpAxisBasicParType AxisParameters;
_LOCAL enum Mechanism_State_ID_enum state_id;

void _INIT ProgramInit(void)
{
	MpAxisBasic_0.Enable     = 1;
	MpAxisBasic_0.MpLink     = &gAxis_Mech_03;
	MpAxisBasic_0.Parameters = &AxisParameters;

	Trajectory_Str.Targets.Position[0] = 700.0;
	Trajectory_Str.Targets.Position[1] = 100.0;
	Trajectory_Str.Targets.Position[2] = 400.0;
	Trajectory_Str.Targets.Position[3] = 600.0;
	Trajectory_Str.Targets.Position[4] = 300.0;

	Trajectory_Str.Targets.Velocity[0] = 500.0;
	Trajectory_Str.Targets.Velocity[1] = 300.0;
	Trajectory_Str.Targets.Velocity[2] = 500.0;
	Trajectory_Str.Targets.Velocity[3] = 100.0;
	Trajectory_Str.Targets.Velocity[4] = 500.0;

	Trajectory_Str.Length = 5;

	state_id = STATE_ID_ACTIVE;
}

void _CYCLIC ProgramCyclic(void)
{
	switch(state_id){
		case STATE_ID_ACTIVE:
			{
				if(Global_MappView_Str.Mech_Id_3.Info.Active == 1){
					state_id = STATE_ID_POWER;
				}
			}
			break;

		case STATE_ID_POWER:
			{
				if(Global_MappView_Str.Mech_Id_3.Info.Power == 1){
					state_id = STATE_ID_HOME;
				}
			}
			break;

		case STATE_ID_HOME:
			{
				if(Global_MappView_Str.Mech_Id_3.Info.Home == 1){
					MpAxisBasic_0.Home = 0;
					Global_MappView_Str.Mech_Id_3.Command.Home = 0;
					state_id = STATE_ID_WAIT;
				}
			}
			break;

		case STATE_ID_WAIT:
			{
				if(Global_MappView_Str.Mech_Id_3.Command.Home == 1){
					state_id = STATE_ID_HOME_UPDATE_PARAMETERS;
				}

				if(Global_MappView_Str.Mech_Id_3.Command.Start == 1){
					Trajectory_Str.Iteration = 0;
					state_id = STATE_ID_UPDATE_PARAMETERS;
				}
			}
			break;

		case STATE_ID_UPDATE_PARAMETERS:
			{
				AxisParameters.Position     = Trajectory_Str.Targets.Position[Trajectory_Str.Iteration];
				AxisParameters.Velocity     = Trajectory_Str.Targets.Velocity[Trajectory_Str.Iteration];
				AxisParameters.Acceleration = Trajectory_Str.Targets.Velocity[Trajectory_Str.Iteration]*10;
				AxisParameters.Deceleration = AxisParameters.Acceleration;

				MpAxisBasic_0.Update = 1;
				if(MpAxisBasic_0.UpdateDone == 1){
					state_id = STATE_ID_MOTION_1;
				}
			}
			break;

		case STATE_ID_MOTION_1:
			{
				MpAxisBasic_0.MoveAbsolute = 1;
				if(MpAxisBasic_0.MoveActive == 1){
					state_id = STATE_ID_MOTION_2;
				}
			}
			break;

		case STATE_ID_MOTION_2:
			{
				if(Global_MappView_Str.Mech_Id_3.Command.Stop == 1){
					state_id = STATE_ID_STOP;
				}else{
					if(MpAxisBasic_0.InPosition == 1 && MpAxisBasic_0.MoveDone == 1){
						MpAxisBasic_0.MoveAbsolute = 0;

						if(Trajectory_Str.Iteration == Trajectory_Str.Length - 1){
							state_id = STATE_ID_WAIT;
						}else{
							Trajectory_Str.Iteration++;
							state_id = STATE_ID_UPDATE_PARAMETERS;
						}
					}
				}
			}
			break;

		case STATE_ID_HOME_UPDATE_PARAMETERS:
			{
				AxisParameters.Position     = 400.0;
				AxisParameters.Velocity     = 250.0;
				AxisParameters.Acceleration = 2500.0;
				AxisParameters.Deceleration = 2500.0;

				MpAxisBasic_0.Update = 1;
				if(MpAxisBasic_0.UpdateDone == 1){
					state_id = STATE_ID_HOME_MOTION_1;
				}
			}
			break;

		case STATE_ID_HOME_MOTION_1:
			{
				MpAxisBasic_0.MoveAbsolute = 1;
				if(MpAxisBasic_0.MoveActive == 1){
					state_id = STATE_ID_HOME_MOTION_2;
				}
			}
			break;

		case STATE_ID_HOME_MOTION_2:
			{
				if(MpAxisBasic_0.InPosition == 1 && MpAxisBasic_0.MoveDone == 1){
					MpAxisBasic_0.MoveAbsolute = 0;
					Global_MappView_Str.Mech_Id_3.Command.Home = 0;
					state_id = STATE_ID_WAIT;
				}
			}
			break;

		case STATE_ID_STOP:
			{
				Global_MappView_Str.Mech_Id_3.Command.Stop  = 0;
				Global_MappView_Str.Mech_Id_3.Command.Start = 0;

				MpAxisBasic_0.MoveAbsolute = 0;
				if(MpAxisBasic_0.MoveActive == 0){
					state_id = STATE_ID_WAIT;
				}
			}
			break;

		case STATE_ID_SAFETY:
			{
			}
			break;

		case STATE_ID_ERROR:
			{
				if(Global_MappView_Str.Mech_Id_3.Info.Error == 1){
					state_id = STATE_ID_WAIT;
				}
			}
			break;

	}

	MpAxisBasic_0.Power      = Global_MappView_Str.Mech_Id_3.Command.Power;
	if(Global_MappView_Str.Mech_Id_3.Command.Home == 1 && Global_MappView_Str.Mech_Id_3.Info.Home == 0){
		MpAxisBasic_0.Home = 1;
	}
	MpAxisBasic_0.ErrorReset = Global_MappView_Str.Mech_Id_3.Command.Reset_Error;

	MpAxisBasic(&MpAxisBasic_0);

	Global_MappView_Str.Mech_Id_3.Info.Active = MpAxisBasic_0.Active;
	Global_MappView_Str.Mech_Id_3.Info.Power  = MpAxisBasic_0.PowerOn;
	Global_MappView_Str.Mech_Id_3.Info.Home   = MpAxisBasic_0.IsHomed;
	Global_MappView_Str.Mech_Id_3.Info.Error  = MpAxisBasic_0.Error;
	Global_MappView_Str.Mech_Id_3.Position = MpAxisBasic_0.Position;

	if(Global_MappView_Str.Mech_Id_3.Info.Error == 1){
		state_id = STATE_ID_ERROR;
	}
}
```

### Program Logical/T_ROB_2_L
